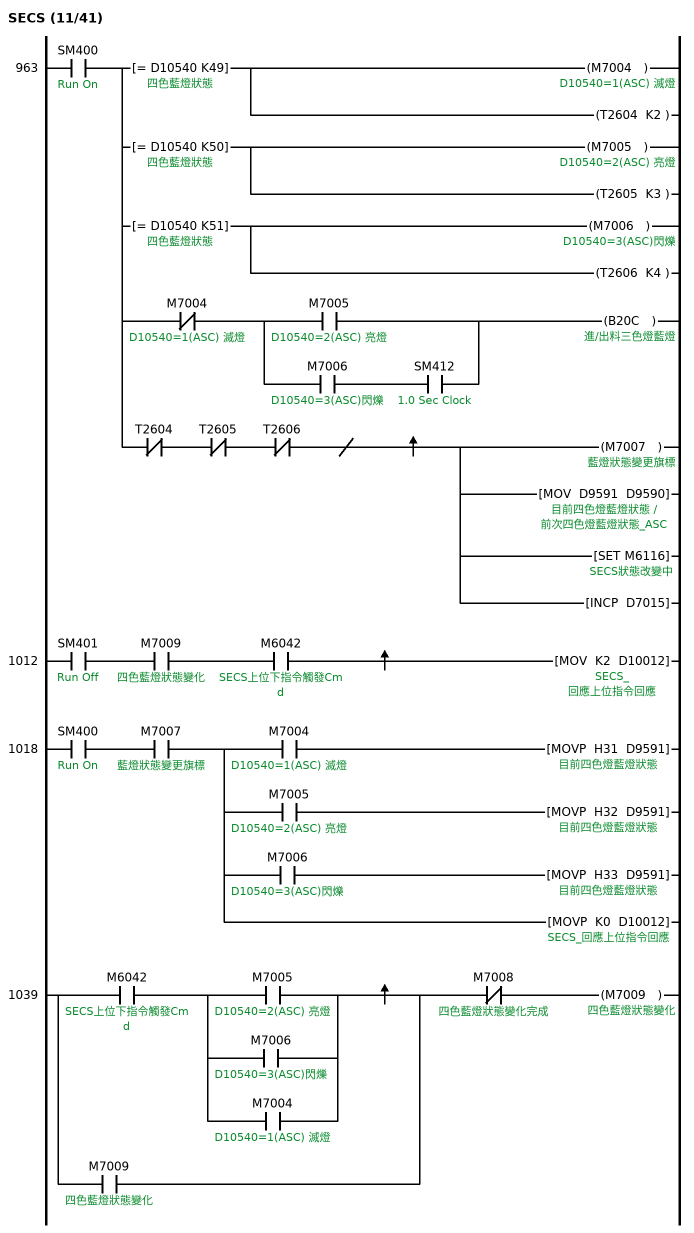
963   LD      SM400  ; Run On
      MPS
      AND=    D10540 K49  ; 四色藍燈狀態
      OUT     M7004  ; D10540=1(ASC) 滅燈
      OUT     T2604 K2
      MRD
      AND=    D10540 K50  ; 四色藍燈狀態
      OUT     M7005  ; D10540=2(ASC) 亮燈
      OUT     T2605 K3
      MRD
      AND=    D10540 K51  ; 四色藍燈狀態
      OUT     M7006  ; D10540=3(ASC)閃爍
      OUT     T2606 K4
      MRD
      ANI     M7004  ; D10540=1(ASC) 滅燈
      LD      M7005  ; D10540=2(ASC) 亮燈
      LD      M7006  ; D10540=3(ASC)閃爍
      AND     SM412  ; 1.0 Sec Clock
      ORB
      ANB
      OUT     B20C  ; 進/出料三色燈藍燈
      MPP
      ANI     T2604
      ANI     T2605
      ANI     T2606
      INV
      MEP
      OUT     M7007  ; 藍燈狀態變更旗標
      MOV     D9591 D9590  ; 目前四色燈藍燈狀態 / 前次四色燈藍燈狀態_ASC
      SET     M6116  ; SECS狀態改變中
      INCP    D7015
1012  LD      SM401  ; Run Off
      AND     M7009  ; 四色藍燈狀態變化
      AND     M6042  ; SECS上位下指令觸發Cmd
      MEP
      MOV     K2 D10012  ; SECS_回應上位指令回應
1018  LD      SM400  ; Run On
      AND     M7007  ; 藍燈狀態變更旗標
      MPS
      AND     M7004  ; D10540=1(ASC) 滅燈
      MOVP    H31 D9591
      MRD
      AND     M7005  ; D10540=2(ASC) 亮燈
      MOVP    H32 D9591
      MRD
      AND     M7006  ; D10540=3(ASC)閃爍
      MOVP    H33 D9591
      MPP
      MOVP    K0 D10012
1039  LD      M6042  ; SECS上位下指令觸發Cmd
      LD      M7005  ; D10540=2(ASC) 亮燈
      OR      M7006  ; D10540=3(ASC)閃爍
      OR      M7004  ; D10540=1(ASC) 滅燈
      ANB
      MEP
      OR      M7009  ; 四色藍燈狀態變化
      ANI     M7008  ; 四色藍燈狀態變化完成
      OUT     M7009  ; 四色藍燈狀態變化
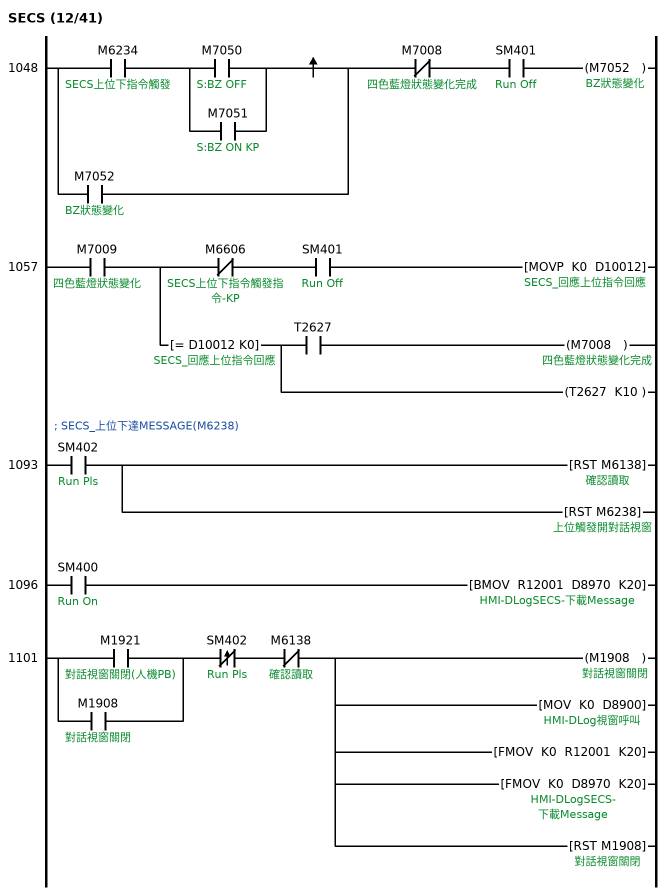
1048  LD      M6234  ; SECS上位下指令觸發
      LD      M7050  ; S:BZ OFF
      OR      M7051  ; S:BZ ON KP
      ANB
      MEP
      OR      M7052  ; BZ狀態變化
      ANI     M7008  ; 四色藍燈狀態變化完成
      AND     SM401  ; Run Off
      OUT     M7052  ; BZ狀態變化
1057  LD      M7009  ; 四色藍燈狀態變化
      MPS
      ANI     M6606  ; SECS上位下指令觸發指令-KP
      AND     SM401  ; Run Off
      MOVP    K0 D10012
      MPP
      AND=    D10012 K0  ; SECS_回應上位指令回應
      MPS
      AND     T2627
      OUT     M7008  ; 四色藍燈狀態變化完成
      MPP
      OUT     T2627 K10
; SECS_上位下達MESSAGE(M6238)
1093  LD      SM402  ; Run Pls
      RST     M6138  ; 確認讀取
      RST     M6238  ; 上位觸發開對話視窗
1096  LD      SM400  ; Run On
      BMOV    R12001 D8970 K20  ; HMI-DLogSECS-下載Message
1101  LD      M1921  ; 對話視窗關閉(人機PB)
      OR      M1908  ; 對話視窗關閉
      ANDPI   SM402  ; Run Pls
      ANI     M6138  ; 確認讀取
      OUT     M1908  ; 對話視窗關閉
      MOV     K0 D8900  ; HMI-DLog視窗呼叫
      FMOV    K0 R12001 K20
      FMOV    K0 D8970 K20
      RST     M1908  ; 對話視窗關閉
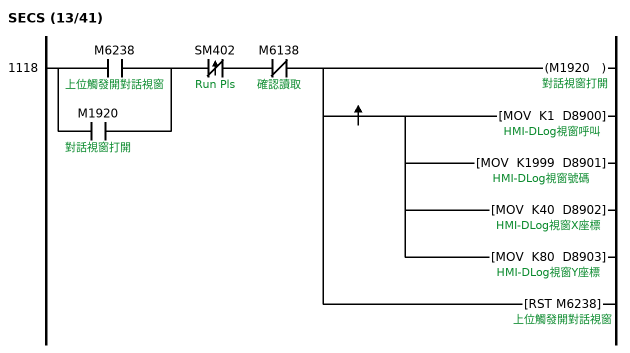
1118  LD      M6238  ; 上位觸發開對話視窗
      OR      M1920  ; 對話視窗打開
      ANDPI   SM402  ; Run Pls
      ANI     M6138  ; 確認讀取
      OUT     M1920  ; 對話視窗打開
      MPS
      MEP
      MOV     K1 D8900
      MOV     K1999 D8901  ; HMI-DLog視窗號碼
      MOV     K40 D8902  ; HMI-DLog視窗X座標
      MOV     K80 D8903  ; HMI-DLog視窗Y座標
      MPP
      RST     M6238  ; 上位觸發開對話視窗
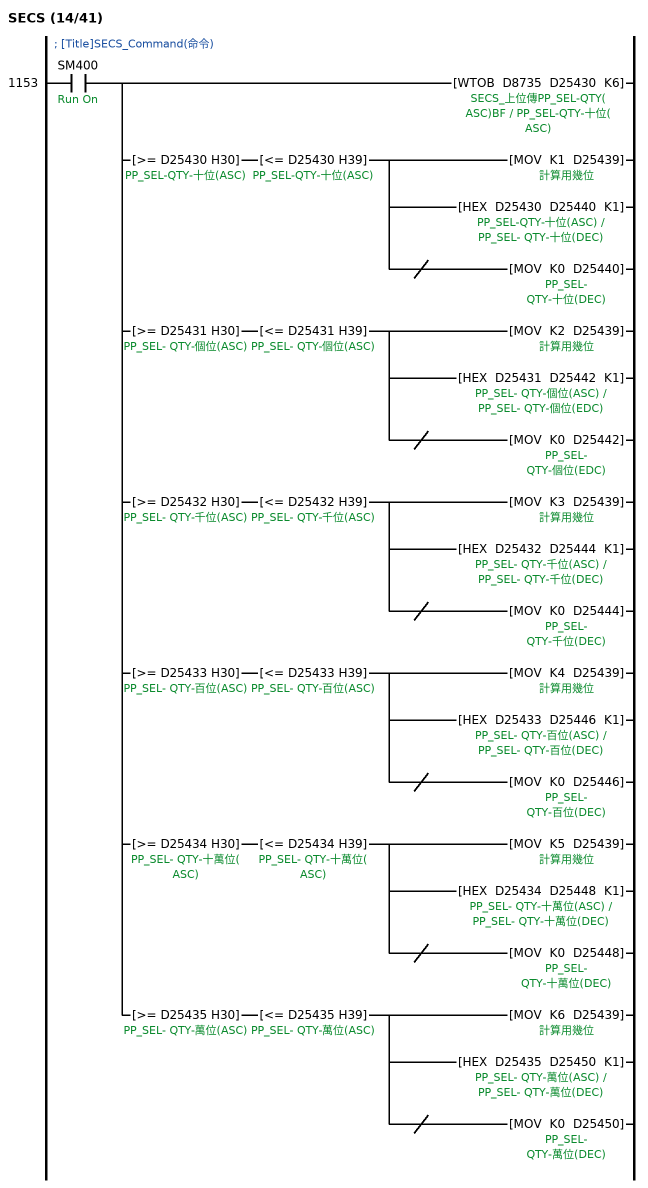
; [Title]SECS_Command(命令)
1153  LD      SM400  ; Run On
      WTOB    D8735 D25430 K6  ; SECS_上位傳PP_SEL-QTY(ASC)BF / PP_SEL-QTY-十位(ASC)
      MPS
      AND>=   D25430 H30  ; PP_SEL-QTY-十位(ASC)
      AND<=   D25430 H39  ; PP_SEL-QTY-十位(ASC)
      MOV     K1 D25439  ; 計算用幾位
      HEX     D25430 D25440 K1  ; PP_SEL- QTY-十位(DEC)
      INV
      MOV     K0 D25440
      MRD
      AND>=   D25431 H30  ; PP_SEL- QTY-個位(ASC)
      AND<=   D25431 H39  ; PP_SEL- QTY-個位(ASC)
      MOV     K2 D25439
      HEX     D25431 D25442 K1  ; PP_SEL- QTY-個位(EDC)
      INV
      MOV     K0 D25442
      MRD
      AND>=   D25432 H30  ; PP_SEL- QTY-千位(ASC)
      AND<=   D25432 H39  ; PP_SEL- QTY-千位(ASC)
      MOV     K3 D25439
      HEX     D25432 D25444 K1  ; PP_SEL- QTY-千位(DEC)
      INV
      MOV     K0 D25444
      MRD
      AND>=   D25433 H30  ; PP_SEL- QTY-百位(ASC)
      AND<=   D25433 H39  ; PP_SEL- QTY-百位(ASC)
      MOV     K4 D25439
      HEX     D25433 D25446 K1  ; PP_SEL- QTY-百位(DEC)
      INV
      MOV     K0 D25446
      MRD
      AND>=   D25434 H30  ; PP_SEL- QTY-十萬位(ASC)
      AND<=   D25434 H39  ; PP_SEL- QTY-十萬位(ASC)
      MOV     K5 D25439
      HEX     D25434 D25448 K1  ; PP_SEL- QTY-十萬位(DEC)
      INV
      MOV     K0 D25448
      MPP
      AND>=   D25435 H30  ; PP_SEL- QTY-萬位(ASC)
      AND<=   D25435 H39  ; PP_SEL- QTY-萬位(ASC)
      MOV     K6 D25439
      HEX     D25435 D25450 K1  ; PP_SEL- QTY-萬位(DEC)
      INV
      MOV     K0 D25450
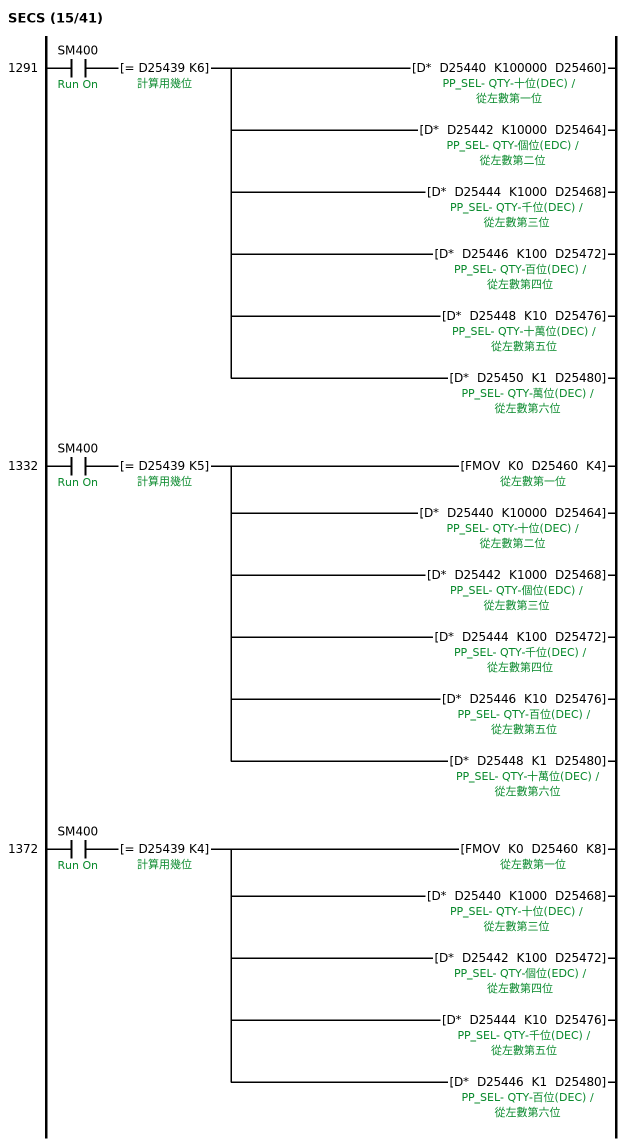
1291  LD      SM400  ; Run On
      AND=    D25439 K6  ; 計算用幾位
      D*      D25440 K100000 D25460  ; 從左數第一位
      D*      D25442 K10000 D25464  ; 從左數第二位
      D*      D25444 K1000 D25468  ; 從左數第三位
      D*      D25446 K100 D25472  ; 從左數第四位
      D*      D25448 K10 D25476  ; 從左數第五位
      D*      D25450 K1 D25480  ; 從左數第六位
1332  LD      SM400  ; Run On
      AND=    D25439 K5  ; 計算用幾位
      FMOV    K0 D25460 K4
      D*      D25440 K10000 D25464
      D*      D25442 K1000 D25468
      D*      D25444 K100 D25472
      D*      D25446 K10 D25476
      D*      D25448 K1 D25480
1372  LD      SM400  ; Run On
      AND=    D25439 K4  ; 計算用幾位
      FMOV    K0 D25460 K8
      D*      D25440 K1000 D25468
      D*      D25442 K100 D25472
      D*      D25444 K10 D25476
      D*      D25446 K1 D25480
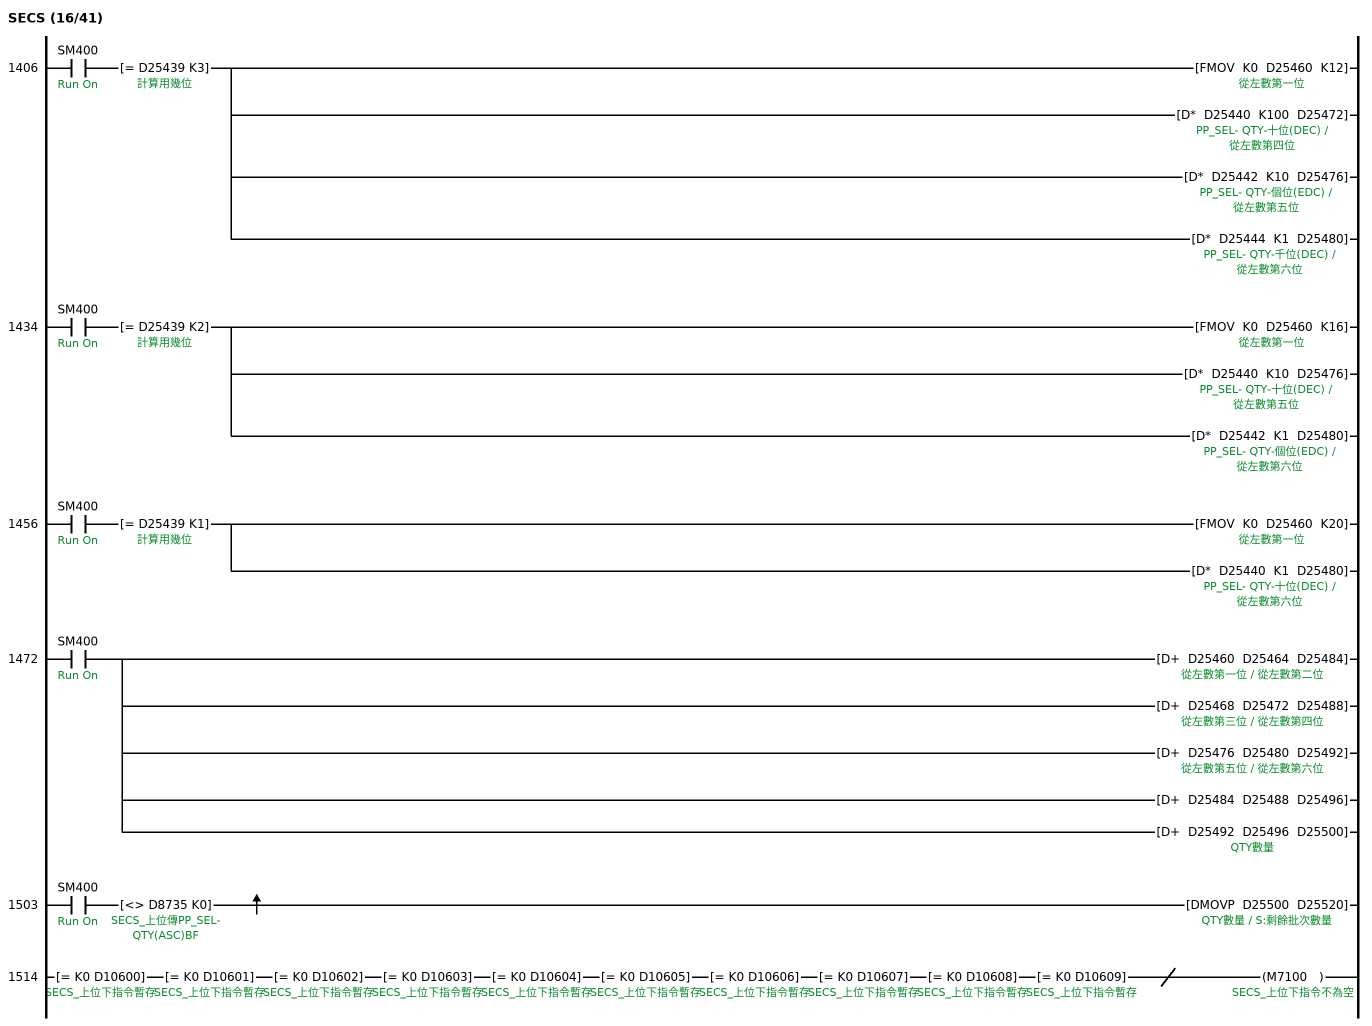
1406  LD      SM400  ; Run On
      AND=    D25439 K3  ; 計算用幾位
      FMOV    K0 D25460 K12
      D*      D25440 K100 D25472
      D*      D25442 K10 D25476
      D*      D25444 K1 D25480
1434  LD      SM400  ; Run On
      AND=    D25439 K2  ; 計算用幾位
      FMOV    K0 D25460 K16
      D*      D25440 K10 D25476
      D*      D25442 K1 D25480
1456  LD      SM400  ; Run On
      AND=    D25439 K1  ; 計算用幾位
      FMOV    K0 D25460 K20
      D*      D25440 K1 D25480
1472  LD      SM400  ; Run On
      D+      D25460 D25464 D25484
      D+      D25468 D25472 D25488
      D+      D25476 D25480 D25492
      D+      D25484 D25488 D25496
      D+      D25492 D25496 D25500  ; QTY數量
1503  LD      SM400  ; Run On
      AND<>   D8735 K0  ; SECS_上位傳PP_SEL-QTY(ASC)BF
      MEP
      DMOVP   D25500 D25520  ; S:剩餘批次數量
1514  LD=     K0 D10600  ; SECS_上位下指令暫存
      AND=    K0 D10601  ; SECS_上位下指令暫存
      AND=    K0 D10602  ; SECS_上位下指令暫存
      AND=    K0 D10603  ; SECS_上位下指令暫存
      AND=    K0 D10604  ; SECS_上位下指令暫存
      AND=    K0 D10605  ; SECS_上位下指令暫存
      AND=    K0 D10606  ; SECS_上位下指令暫存
      AND=    K0 D10607  ; SECS_上位下指令暫存
      AND=    K0 D10608  ; SECS_上位下指令暫存
      AND=    K0 D10609  ; SECS_上位下指令暫存
      INV
      OUT     M7100  ; SECS_上位下指令不為空
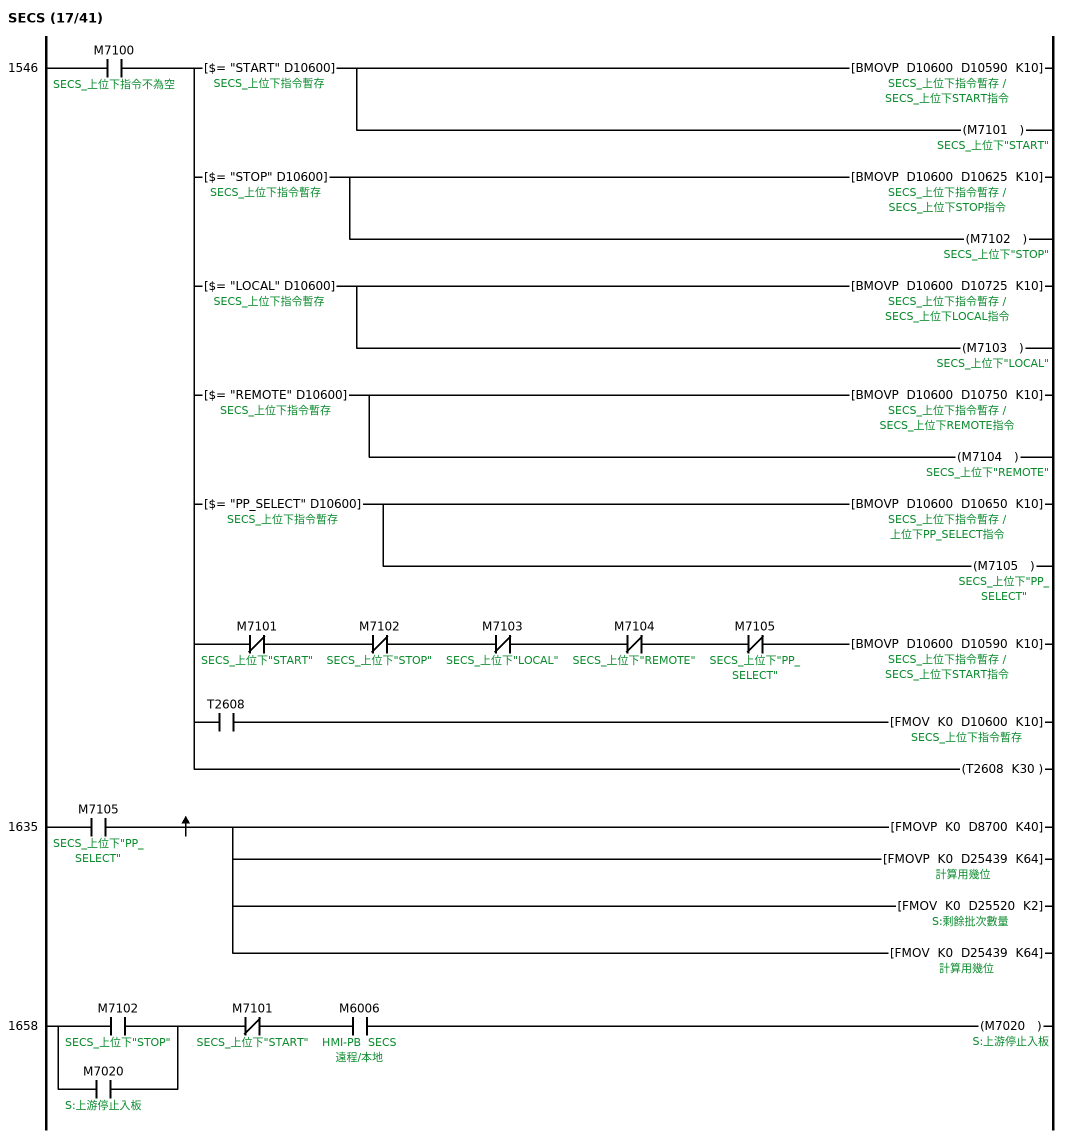
1546  LD      M7100  ; SECS_上位下指令不為空
      MPS
      AND$=   "START" D10600  ; SECS_上位下指令暫存
      BMOVP   D10600 D10590 K10  ; SECS_上位下START指令
      OUT     M7101  ; SECS_上位下"START"
      MRD
      AND$=   "STOP" D10600  ; SECS_上位下指令暫存
      BMOVP   D10600 D10625 K10  ; SECS_上位下STOP指令
      OUT     M7102  ; SECS_上位下"STOP"
      MRD
      AND$=   "LOCAL" D10600  ; SECS_上位下指令暫存
      BMOVP   D10600 D10725 K10  ; SECS_上位下LOCAL指令
      OUT     M7103  ; SECS_上位下"LOCAL"
      MRD
      AND$=   "REMOTE" D10600  ; SECS_上位下指令暫存
      BMOVP   D10600 D10750 K10  ; SECS_上位下REMOTE指令
      OUT     M7104  ; SECS_上位下"REMOTE"
      MRD
      AND$=   "PP_SELECT" D10600  ; SECS_上位下指令暫存
      BMOVP   D10600 D10650 K10  ; 上位下PP_SELECT指令
      OUT     M7105  ; SECS_上位下"PP_SELECT"
      MRD
      ANI     M7101  ; SECS_上位下"START"
      ANI     M7102  ; SECS_上位下"STOP"
      ANI     M7103  ; SECS_上位下"LOCAL"
      ANI     M7104  ; SECS_上位下"REMOTE"
      ANI     M7105  ; SECS_上位下"PP_SELECT"
      BMOVP   D10600 D10590 K10
      MRD
      AND     T2608
      FMOV    K0 D10600 K10
      MPP
      OUT     T2608 K30
1635  LD      M7105  ; SECS_上位下"PP_SELECT"
      MEP
      FMOVP   K0 D8700 K40
      FMOVP   K0 D25439 K64
      FMOV    K0 D25520 K2
      FMOV    K0 D25439 K64
1658  LD      M7102  ; SECS_上位下"STOP"
      OR      M7020  ; S:上游停止入板
      ANI     M7101  ; SECS_上位下"START"
      AND     M6006  ; HMI-PB  SECS  遠程/本地
      OUT     M7020  ; S:上游停止入板
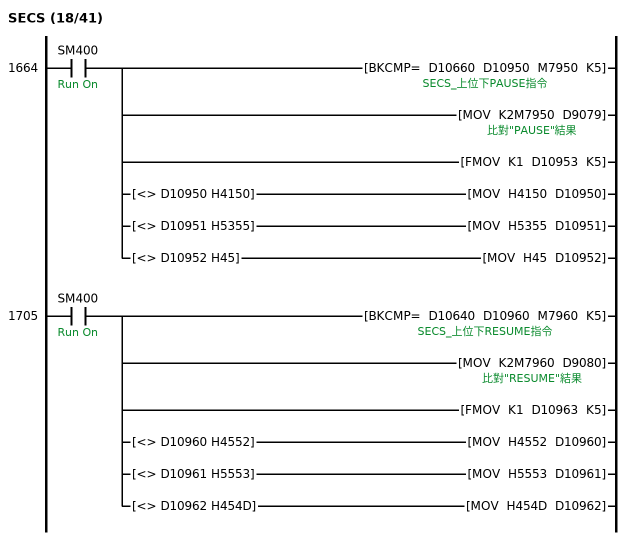
1664  LD      SM400  ; Run On
      BKCMP=  D10660 D10950 M7950 K5  ; SECS_上位下PAUSE指令
        [note] 上位下PAUSE指令
      MOV     K2M7950 D9079  ; 比對"PAUSE"結果
      FMOV    K1 D10953 K5
      MPS
      AND<>   D10950 H4150
      MOV     H4150 D10950
      MRD
      AND<>   D10951 H5355
      MOV     H5355 D10951
      MPP
      AND<>   D10952 H45
      MOV     H45 D10952
1705  LD      SM400  ; Run On
      BKCMP=  D10640 D10960 M7960 K5  ; SECS_上位下RESUME指令
        [note] 上位下RESUME指令
      MOV     K2M7960 D9080  ; 比對"RESUME"結果
      FMOV    K1 D10963 K5
      MPS
      AND<>   D10960 H4552
      MOV     H4552 D10960
      MRD
      AND<>   D10961 H5553
      MOV     H5553 D10961
      MPP
      AND<>   D10962 H454D
      MOV     H454D D10962
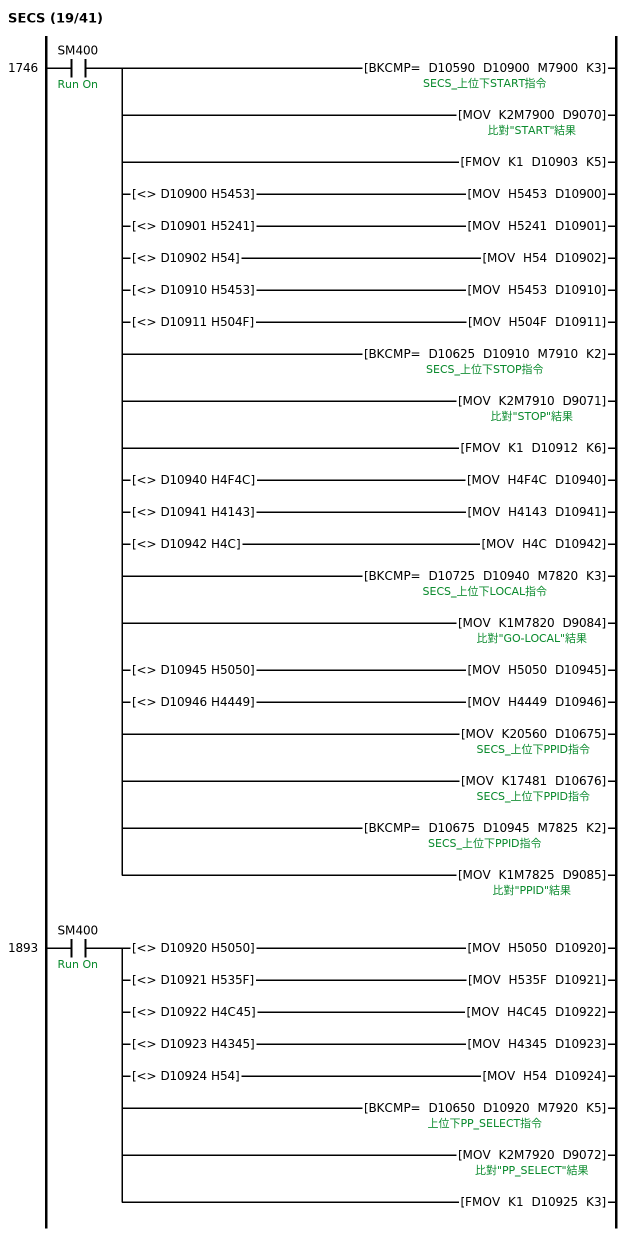
1746  LD      SM400  ; Run On
      BKCMP=  D10590 D10900 M7900 K3
        [note] 上位下START指令
      MOV     K2M7900 D9070  ; 比對"START"結果
      FMOV    K1 D10903 K5
      MPS
      AND<>   D10900 H5453
      MOV     H5453 D10900
      MRD
      AND<>   D10901 H5241
      MOV     H5241 D10901
      MRD
      AND<>   D10902 H54
      MOV     H54 D10902
      MRD
      AND<>   D10910 H5453
      MOV     H5453 D10910
      MRD
      AND<>   D10911 H504F
      MOV     H504F D10911
      MPP
      BKCMP=  D10625 D10910 M7910 K2
        [note] 上位下STOP指令
      MOV     K2M7910 D9071  ; 比對"STOP"結果
      FMOV    K1 D10912 K6
      MPS
      AND<>   D10940 H4F4C
      MOV     H4F4C D10940
      MRD
      AND<>   D10941 H4143
      MOV     H4143 D10941
      MRD
      AND<>   D10942 H4C
      MOV     H4C D10942
      MPP
      BKCMP=  D10725 D10940 M7820 K3
        [note] 上位下GO-LOCAL指令
      MOV     K1M7820 D9084  ; 比對"GO-LOCAL"結果
      MPS
      AND<>   D10945 H5050
      MOV     H5050 D10945
      MRD
      AND<>   D10946 H4449
      MOV     H4449 D10946
      MPP
      MOV     K20560 D10675  ; SECS_上位下PPID指令
      MOV     K17481 D10676  ; SECS_上位下PPID指令
      BKCMP=  D10675 D10945 M7825 K2
        [note] 上位下PPID指令
      MOV     K1M7825 D9085  ; 比對"PPID"結果
1893  LD      SM400  ; Run On
      MPS
      AND<>   D10920 H5050
      MOV     H5050 D10920
      MRD
      AND<>   D10921 H535F
      MOV     H535F D10921
      MRD
      AND<>   D10922 H4C45
      MOV     H4C45 D10922
      MRD
      AND<>   D10923 H4345
      MOV     H4345 D10923
      MRD
      AND<>   D10924 H54
      MOV     H54 D10924
      MPP
      BKCMP=  D10650 D10920 M7920 K5
        [note] 上位下PP_SELECT指令
      MOV     K2M7920 D9072  ; 比對"PP_SELECT"結果
      FMOV    K1 D10925 K3
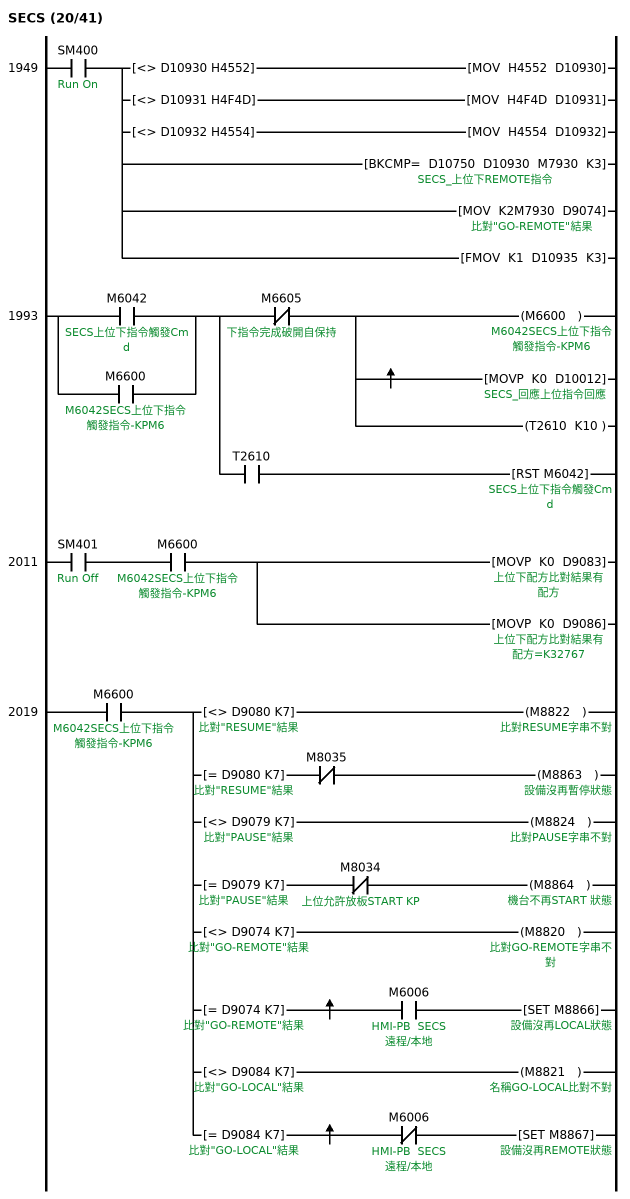
1949  LD      SM400  ; Run On
      MPS
      AND<>   D10930 H4552
      MOV     H4552 D10930
      MRD
      AND<>   D10931 H4F4D
      MOV     H4F4D D10931
      MRD
      AND<>   D10932 H4554
      MOV     H4554 D10932
      MPP
      BKCMP=  D10750 D10930 M7930 K3
        [note] 上位下GO-REMOTE指令
      MOV     K2M7930 D9074  ; 比對"GO-REMOTE"結果
      FMOV    K1 D10935 K3
1993  LD      M6042  ; SECS上位下指令觸發Cmd
      OR      M6600  ; M6042SECS上位下指令觸發指令-KPM6
      MPS
      ANI     M6605  ; 下指令完成破開自保持
      OUT     M6600  ; M6042SECS上位下指令觸發指令-KPM6
      MPS
      MEP
      MOVP    K0 D10012
      MPP
      OUT     T2610 K10
      MPP
      AND     T2610
      RST     M6042  ; SECS上位下指令觸發Cmd
2011  LD      SM401  ; Run Off
      AND     M6600  ; M6042SECS上位下指令觸發指令-KPM6
      MOVP    K0 D9083  ; 上位下配方比對結果有配方
      MOVP    K0 D9086  ; 上位下配方比對結果有配方=K32767
2019  LD      M6600  ; M6042SECS上位下指令觸發指令-KPM6
      MPS
      AND<>   D9080 K7  ; 比對"RESUME"結果
      OUT     M8822  ; 比對RESUME字串不對
      MRD
      AND=    D9080 K7  ; 比對"RESUME"結果
      ANI     M8035
      OUT     M8863  ; 設備沒再暫停狀態
      MRD
      AND<>   D9079 K7  ; 比對"PAUSE"結果
      OUT     M8824  ; 比對PAUSE字串不對
      MRD
      AND=    D9079 K7  ; 比對"PAUSE"結果
      ANI     M8034  ; 上位允許放板START KP
      OUT     M8864  ; 機台不再START 狀態
      MRD
      AND<>   D9074 K7  ; 比對"GO-REMOTE"結果
      OUT     M8820  ; 比對GO-REMOTE字串不對
      MRD
      AND=    D9074 K7  ; 比對"GO-REMOTE"結果
      MEP
      AND     M6006  ; HMI-PB  SECS  遠程/本地
      SET     M8866  ; 設備沒再LOCAL狀態
      MRD
      AND<>   D9084 K7  ; 比對"GO-LOCAL"結果
      OUT     M8821  ; 名稱GO-LOCAL比對不對
      MPP
      AND=    D9084 K7  ; 比對"GO-LOCAL"結果
      MEP
      ANI     M6006  ; HMI-PB  SECS  遠程/本地
      SET     M8867  ; 設備沒再REMOTE狀態
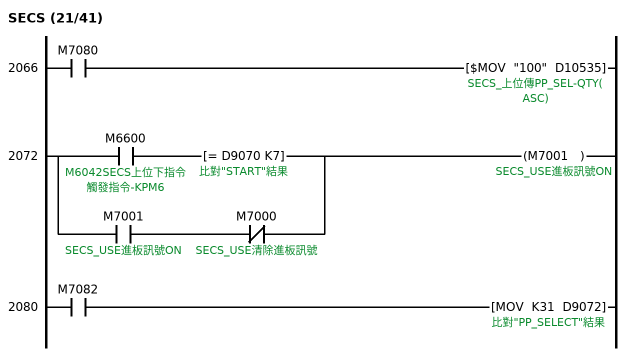
2066  LD      M7080
      $MOV    "100" D10535  ; SECS_上位傳PP_SEL-QTY(ASC)
2072  LD      M6600  ; M6042SECS上位下指令觸發指令-KPM6
      AND=    D9070 K7  ; 比對"START"結果
      LD      M7001  ; SECS_USE進板訊號ON
      ANI     M7000  ; SECS_USE清除進板訊號
      ORB
      OUT     M7001  ; SECS_USE進板訊號ON
2080  LD      M7082
      MOV     K31 D9072
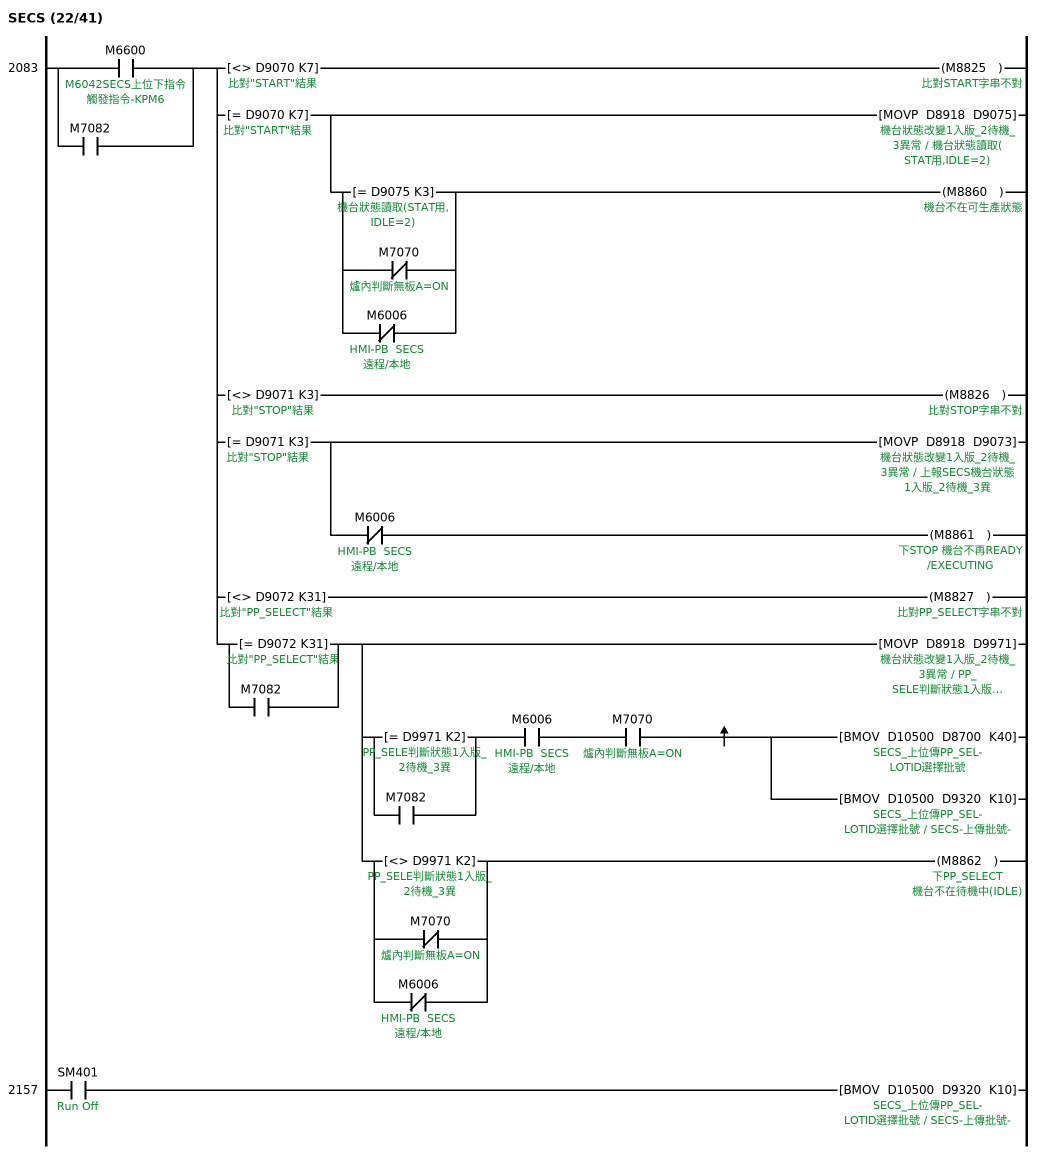
2083  LD      M6600  ; M6042SECS上位下指令觸發指令-KPM6
      OR      M7082
      MPS
      AND<>   D9070 K7  ; 比對"START"結果
      OUT     M8825  ; 比對START字串不對
      MRD
      AND=    D9070 K7  ; 比對"START"結果
      MOVP    D8918 D9075  ; 機台狀態讀取(STAT用,IDLE=2)
      LD=     D9075 K3  ; 機台狀態讀取(STAT用,IDLE=2)
      ORI     M7070  ; 爐內判斷無板A=ON
      ORI     M6006  ; HMI-PB  SECS  遠程/本地
      ANB
      OUT     M8860  ; 機台不在可生產狀態
      MRD
      AND<>   D9071 K3  ; 比對"STOP"結果
      OUT     M8826  ; 比對STOP字串不對
      MRD
      AND=    D9071 K3  ; 比對"STOP"結果
      MOVP    D8918 D9073  ; 上報SECS機台狀態1入版_2待機_3異
      ANI     M6006  ; HMI-PB  SECS  遠程/本地
      OUT     M8861  ; 下STOP 機台不再READY/EXECUTING
      MRD
      AND<>   D9072 K31  ; 比對"PP_SELECT"結果
      OUT     M8827  ; 比對PP_SELECT字串不對
      MPP
      LD=     D9072 K31  ; 比對"PP_SELECT"結果
      OR      M7082
      ANB
      MOVP    D8918 D9971  ; PP_SELE判斷狀態1入版_2待機_3異
      MPS
      LD=     D9971 K2  ; PP_SELE判斷狀態1入版_2待機_3異
      OR      M7082
      ANB
      AND     M6006  ; HMI-PB  SECS  遠程/本地
      AND     M7070  ; 爐內判斷無板A=ON
      MEP
      BMOV    D10500 D8700 K40  ; SECS_上位傳PP_SEL-LOTID選擇批號
      BMOV    D10500 D9320 K10  ; SECS-上傳批號-
      MPP
      LD<>    D9971 K2  ; PP_SELE判斷狀態1入版_2待機_3異
      ORI     M7070  ; 爐內判斷無板A=ON
      ORI     M6006  ; HMI-PB  SECS  遠程/本地
      ANB
      OUT     M8862  ; 下PP_SELECT 機台不在待機中(IDLE)
2157  LD      SM401  ; Run Off
      BMOV    D10500 D9320 K10
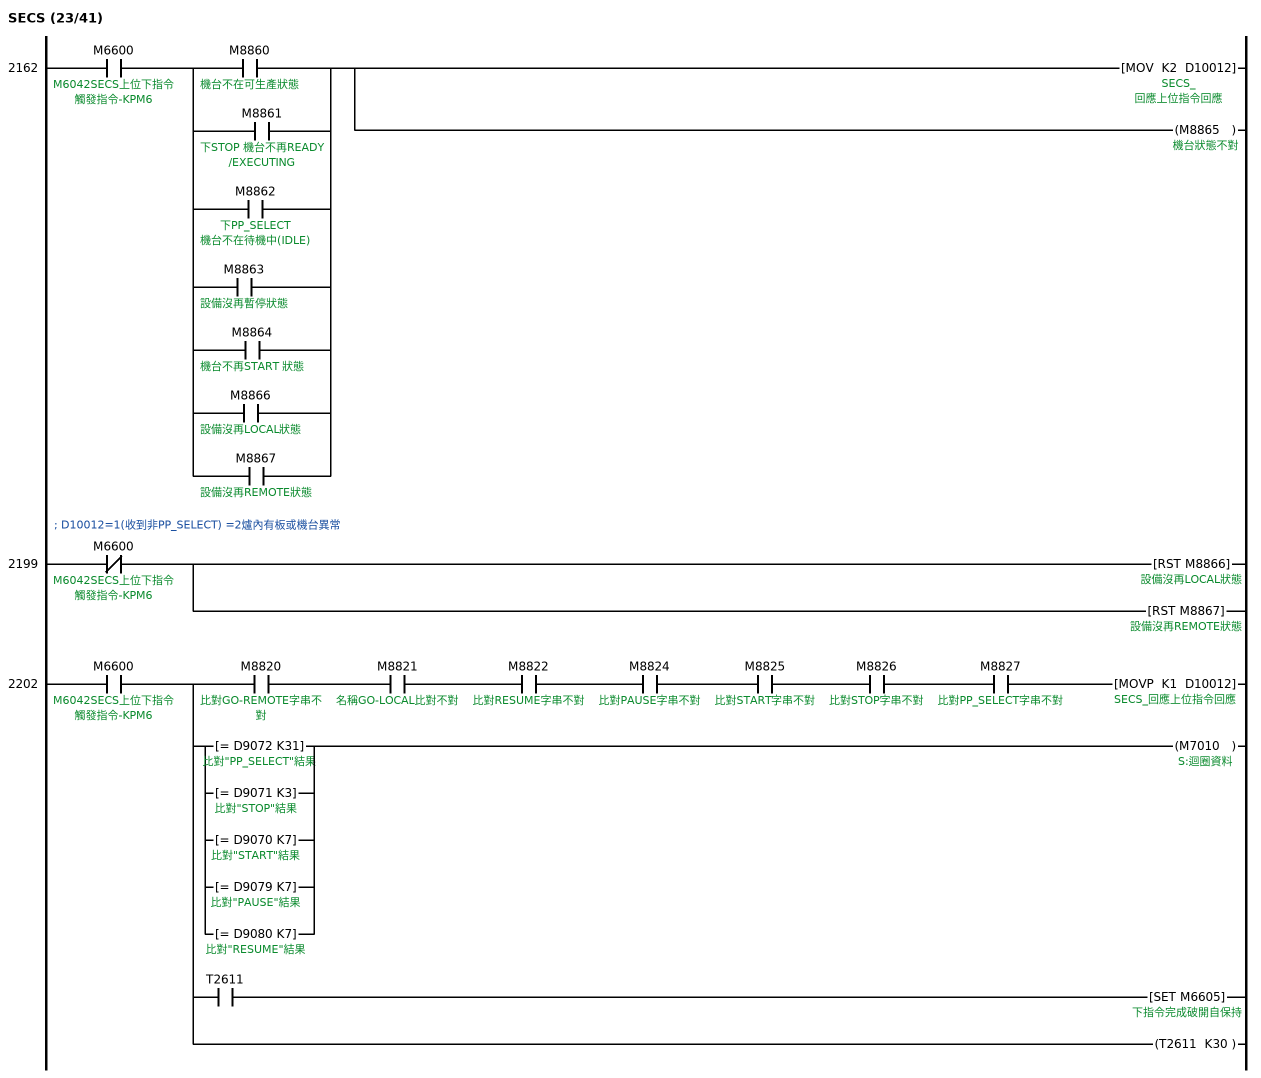
2162  LD      M6600  ; M6042SECS上位下指令觸發指令-KPM6
      LD      M8860  ; 機台不在可生產狀態
      OR      M8861  ; 下STOP 機台不再READY/EXECUTING
      OR      M8862  ; 下PP_SELECT 機台不在待機中(IDLE)
      OR      M8863  ; 設備沒再暫停狀態
      OR      M8864  ; 機台不再START 狀態
      OR      M8866  ; 設備沒再LOCAL狀態
      OR      M8867  ; 設備沒再REMOTE狀態
      ANB
      MOV     K2 D10012
      OUT     M8865  ; 機台狀態不對
; D10012=1(收到非PP_SELECT) =2爐內有板或機台異常
2199  LDI     M6600  ; M6042SECS上位下指令觸發指令-KPM6
      RST     M8866  ; 設備沒再LOCAL狀態
      RST     M8867  ; 設備沒再REMOTE狀態
2202  LD      M6600  ; M6042SECS上位下指令觸發指令-KPM6
      MPS
      AND     M8820  ; 比對GO-REMOTE字串不對
      AND     M8821  ; 名稱GO-LOCAL比對不對
      AND     M8822  ; 比對RESUME字串不對
      AND     M8824  ; 比對PAUSE字串不對
      AND     M8825  ; 比對START字串不對
      AND     M8826  ; 比對STOP字串不對
      AND     M8827  ; 比對PP_SELECT字串不對
      MOVP    K1 D10012
      MRD
      LD=     D9072 K31  ; 比對"PP_SELECT"結果
      OR=     D9071 K3  ; 比對"STOP"結果
      OR=     D9070 K7  ; 比對"START"結果
      OR=     D9079 K7  ; 比對"PAUSE"結果
      OR=     D9080 K7  ; 比對"RESUME"結果
      ANB
      OUT     M7010  ; S:迴圈資料
      MRD
      AND     T2611
      SET     M6605  ; 下指令完成破開自保持
      MPP
      OUT     T2611 K30
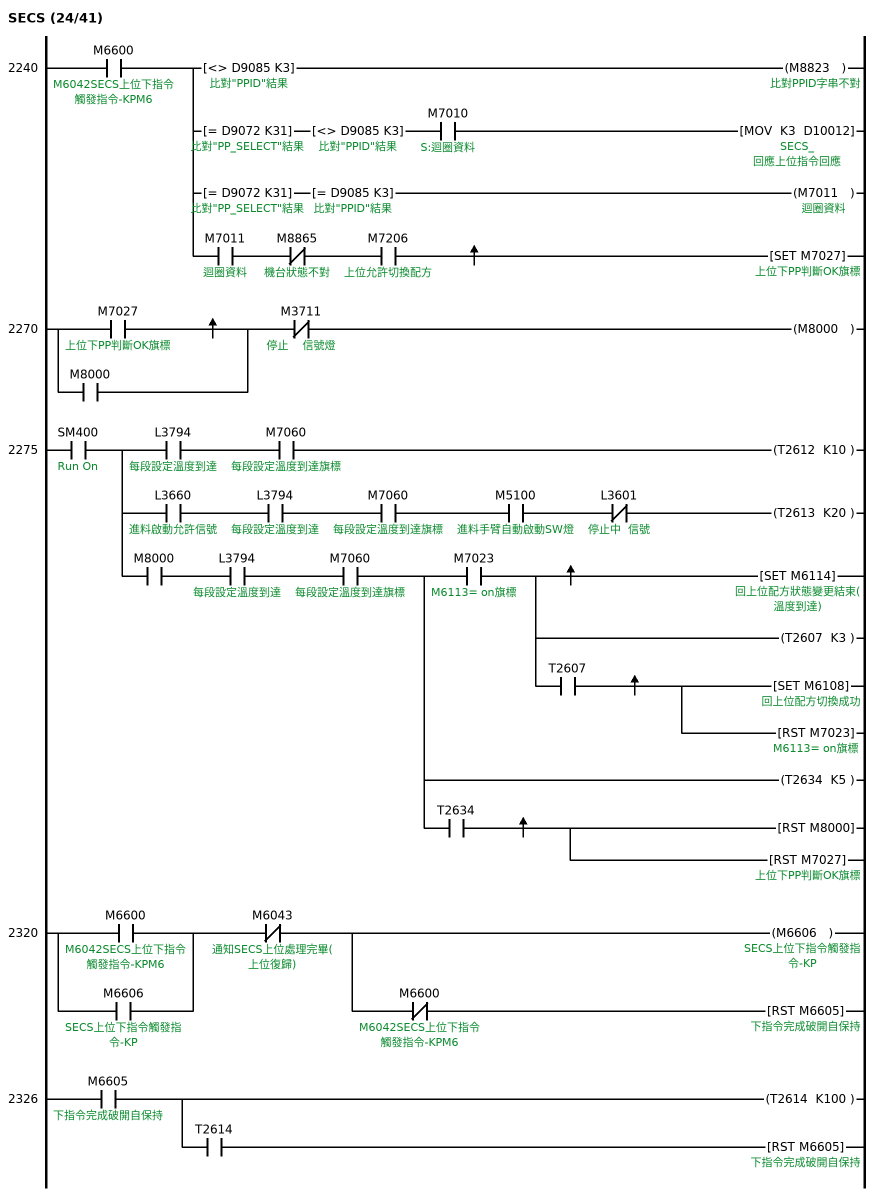
2240  LD      M6600  ; M6042SECS上位下指令觸發指令-KPM6
      MPS
      AND<>   D9085 K3  ; 比對"PPID"結果
      OUT     M8823  ; 比對PPID字串不對
      MRD
      AND=    D9072 K31  ; 比對"PP_SELECT"結果
      AND<>   D9085 K3  ; 比對"PPID"結果
      AND     M7010  ; S:迴圈資料
      MOV     K3 D10012
      MRD
      AND=    D9072 K31  ; 比對"PP_SELECT"結果
      AND=    D9085 K3  ; 比對"PPID"結果
      OUT     M7011  ; 迴圈資料
      MPP
      AND     M7011  ; 迴圈資料
      ANI     M8865  ; 機台狀態不對
      AND     M7206  ; 上位允許切換配方
      MEP
      SET     M7027  ; 上位下PP判斷OK旗標
2270  LD      M7027  ; 上位下PP判斷OK旗標
      MEP
      OR      M8000
      ANI     M3711  ; 停止    信號燈
      OUT     M8000
2275  LD      SM400  ; Run On
      MPS
      AND     L3794  ; 每段設定溫度到達
      AND     M7060  ; 每段設定溫度到達旗標
      OUT     T2612 K10
      MRD
      AND     L3660  ; 進料啟動允許信號
      AND     L3794  ; 每段設定溫度到達
      AND     M7060  ; 每段設定溫度到達旗標
      AND     M5100  ; 進料手臂自動啟動SW燈
      ANI     L3601  ; 停止中  信號
      OUT     T2613 K20
      MPP
      AND     M8000
      AND     L3794  ; 每段設定溫度到達
      AND     M7060  ; 每段設定溫度到達旗標
      MPS
      AND     M7023  ; M6113= on旗標
      MPS
      MEP
      SET     M6114  ; 回上位配方狀態變更結束(溫度到達)
      MPP
      OUT     T2607 K3
      AND     T2607
      MEP
      SET     M6108  ; 回上位配方切換成功
      RST     M7023  ; M6113= on旗標
      MPP
      OUT     T2634 K5
      AND     T2634
      MEP
      RST     M8000
      RST     M7027  ; 上位下PP判斷OK旗標
2320  LD      M6600  ; M6042SECS上位下指令觸發指令-KPM6
      OR      M6606  ; SECS上位下指令觸發指令-KP
      ANI     M6043  ; 通知SECS上位處理完畢(上位復歸)
      OUT     M6606  ; SECS上位下指令觸發指令-KP
      ANI     M6600  ; M6042SECS上位下指令觸發指令-KPM6
      RST     M6605  ; 下指令完成破開自保持
2326  LD      M6605  ; 下指令完成破開自保持
      OUT     T2614 K100
      AND     T2614
      RST     M6605  ; 下指令完成破開自保持
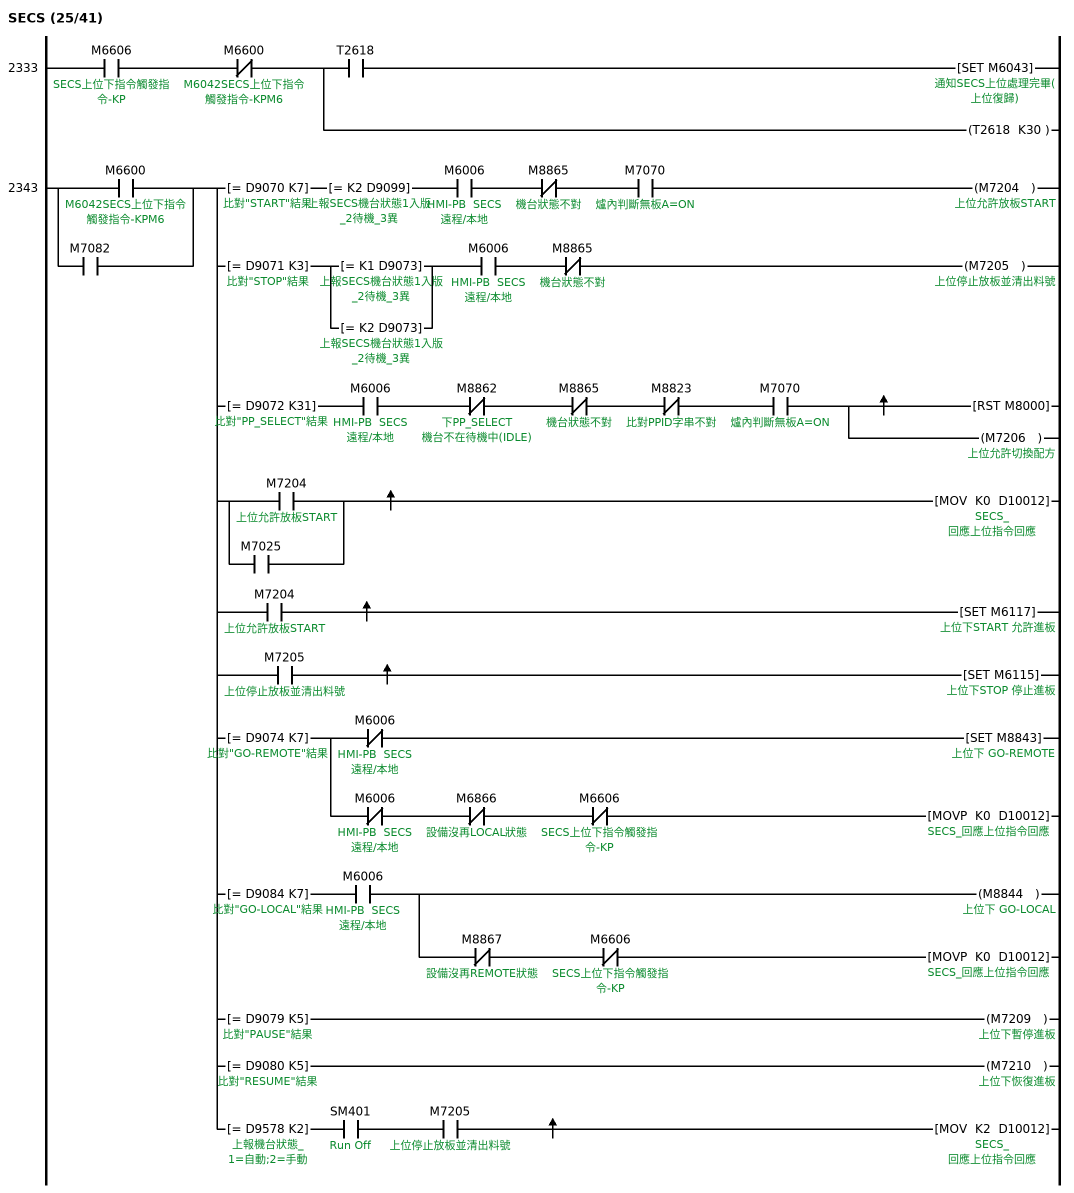
2333  LD      M6606  ; SECS上位下指令觸發指令-KP
      ANI     M6600  ; M6042SECS上位下指令觸發指令-KPM6
      MPS
      AND     T2618
      SET     M6043  ; 通知SECS上位處理完畢(上位復歸)
      MPP
      OUT     T2618 K30
2343  LD      M6600  ; M6042SECS上位下指令觸發指令-KPM6
      OR      M7082
      MPS
      AND=    D9070 K7  ; 比對"START"結果
      AND=    K2 D9099  ; 上報SECS機台狀態1入版_2待機_3異
      AND     M6006  ; HMI-PB  SECS  遠程/本地
      ANI     M8865  ; 機台狀態不對
      AND     M7070  ; 爐內判斷無板A=ON
      OUT     M7204  ; 上位允許放板START
      MRD
      AND=    D9071 K3  ; 比對"STOP"結果
      LD=     K1 D9073  ; 上報SECS機台狀態1入版_2待機_3異
      OR=     K2 D9073  ; 上報SECS機台狀態1入版_2待機_3異
      ANB
      AND     M6006  ; HMI-PB  SECS  遠程/本地
      ANI     M8865  ; 機台狀態不對
      OUT     M7205  ; 上位停止放板並清出料號
      MRD
      AND=    D9072 K31  ; 比對"PP_SELECT"結果
      AND     M6006  ; HMI-PB  SECS  遠程/本地
      ANI     M8862  ; 下PP_SELECT 機台不在待機中(IDLE)
      ANI     M8865  ; 機台狀態不對
      ANI     M8823  ; 比對PPID字串不對
      AND     M7070  ; 爐內判斷無板A=ON
      MPS
      MEP
      RST     M8000
      MPP
      OUT     M7206  ; 上位允許切換配方
      MRD
      LD      M7204  ; 上位允許放板START
      OR      M7025
      ANB
      MEP
      MOV     K0 D10012
      MRD
      AND     M7204  ; 上位允許放板START
      MEP
      SET     M6117  ; 上位下START 允許進板
      MRD
      AND     M7205  ; 上位停止放板並清出料號
      MEP
      SET     M6115  ; 上位下STOP 停止進板
      MRD
      AND=    D9074 K7  ; 比對"GO-REMOTE"結果
      MPS
      ANI     M6006  ; HMI-PB  SECS  遠程/本地
      SET     M8843  ; 上位下 GO-REMOTE
      MPP
      ANI     M6006  ; HMI-PB  SECS  遠程/本地
      ANI     M6866  ; 設備沒再LOCAL狀態
      ANI     M6606  ; SECS上位下指令觸發指令-KP
      MOVP    K0 D10012
      MRD
      AND=    D9084 K7  ; 比對"GO-LOCAL"結果
      AND     M6006  ; HMI-PB  SECS  遠程/本地
      OUT     M8844  ; 上位下 GO-LOCAL
      ANI     M8867  ; 設備沒再REMOTE狀態
      ANI     M6606  ; SECS上位下指令觸發指令-KP
      MOVP    K0 D10012
      MRD
      AND=    D9079 K5  ; 比對"PAUSE"結果
      OUT     M7209  ; 上位下暫停進板
      MRD
      AND=    D9080 K5  ; 比對"RESUME"結果
      OUT     M7210  ; 上位下恢復進板
      MPP
      AND=    D9578 K2  ; 上報機台狀態_1=自動;2=手動
      AND     SM401  ; Run Off
      AND     M7205  ; 上位停止放板並清出料號
      MEP
      MOV     K2 D10012
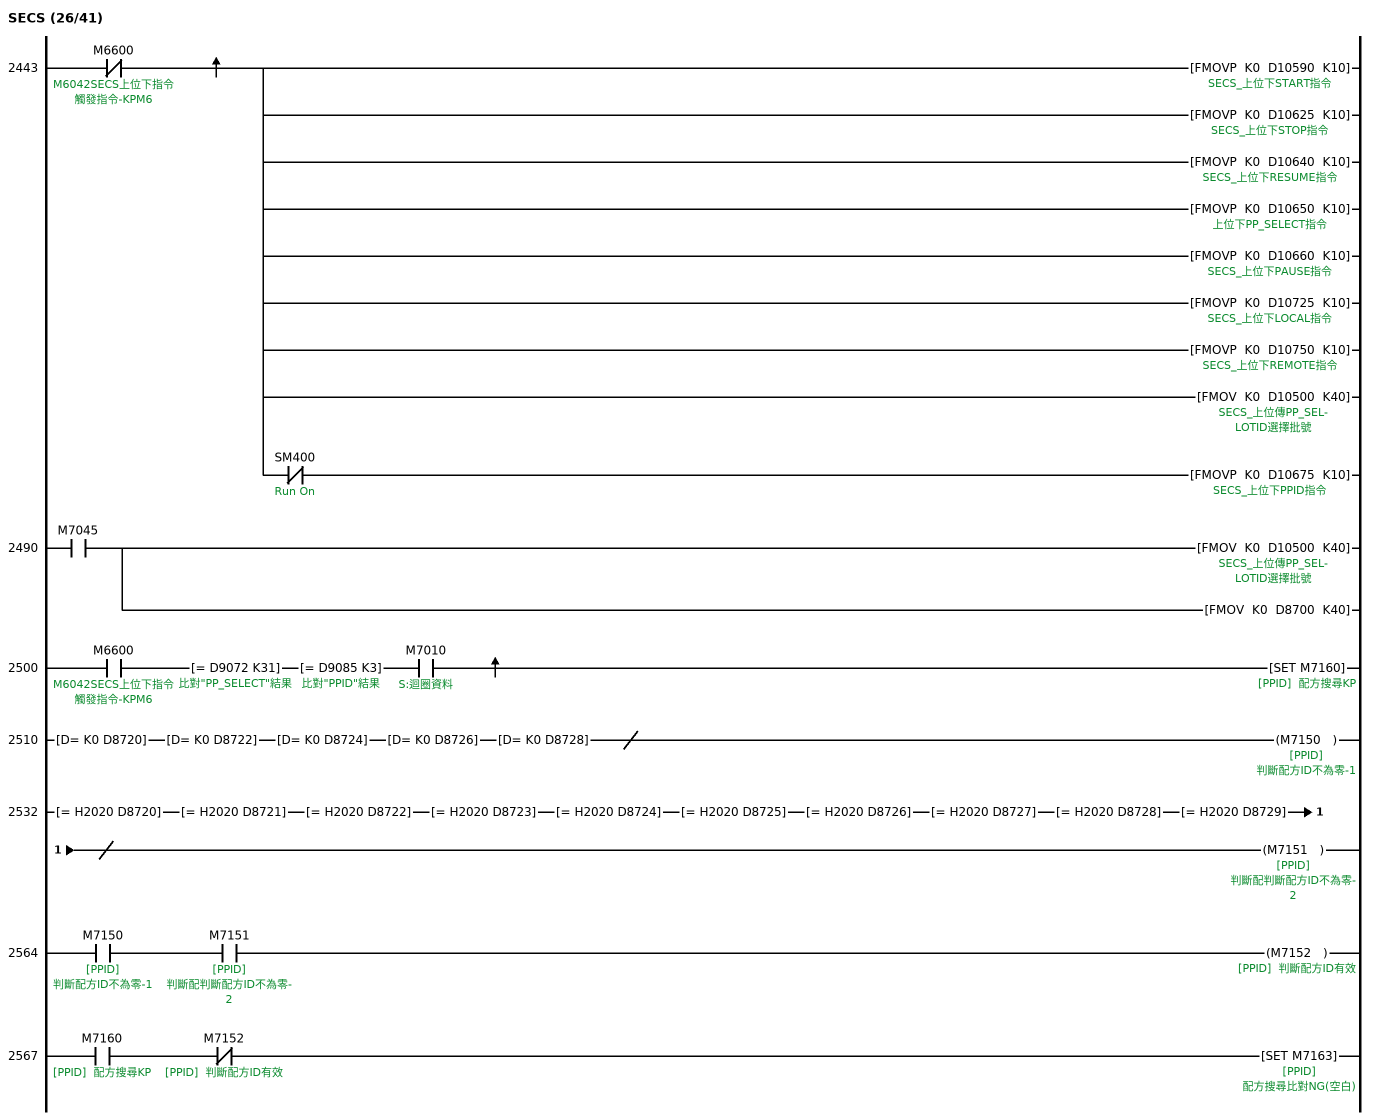
2443  LDI     M6600  ; M6042SECS上位下指令觸發指令-KPM6
      MEP
      FMOVP   K0 D10590 K10
      FMOVP   K0 D10625 K10
      FMOVP   K0 D10640 K10
      FMOVP   K0 D10650 K10
      FMOVP   K0 D10660 K10
      FMOVP   K0 D10725 K10
      FMOVP   K0 D10750 K10
      FMOV    K0 D10500 K40
      ANI     SM400  ; Run On
      FMOVP   K0 D10675 K10
2490  LD      M7045
      FMOV    K0 D10500 K40
      FMOV    K0 D8700 K40
2500  LD      M6600  ; M6042SECS上位下指令觸發指令-KPM6
      AND=    D9072 K31  ; 比對"PP_SELECT"結果
      AND=    D9085 K3  ; 比對"PPID"結果
      AND     M7010  ; S:迴圈資料
      MEP
      SET     M7160  ; [PPID]  配方搜尋KP
2510  LDD=    K0 D8720
      ANDD=   K0 D8722
      ANDD=   K0 D8724
      ANDD=   K0 D8726
      ANDD=   K0 D8728
      INV
      OUT     M7150  ; [PPID]  判斷配方ID不為零-1
2532  LD=     H2020 D8720
      AND=    H2020 D8721
      AND=    H2020 D8722
      AND=    H2020 D8723
      AND=    H2020 D8724
      AND=    H2020 D8725
      AND=    H2020 D8726
      AND=    H2020 D8727
      AND=    H2020 D8728
      AND=    H2020 D8729
      INV
      OUT     M7151  ; [PPID]  判斷配判斷配方ID不為零-2
2564  LD      M7150  ; [PPID]  判斷配方ID不為零-1
      AND     M7151  ; [PPID]  判斷配判斷配方ID不為零-2
      OUT     M7152  ; [PPID]  判斷配方ID有效
2567  LD      M7160  ; [PPID]  配方搜尋KP
      ANI     M7152  ; [PPID]  判斷配方ID有效
      SET     M7163  ; [PPID]  配方搜尋比對NG(空白)
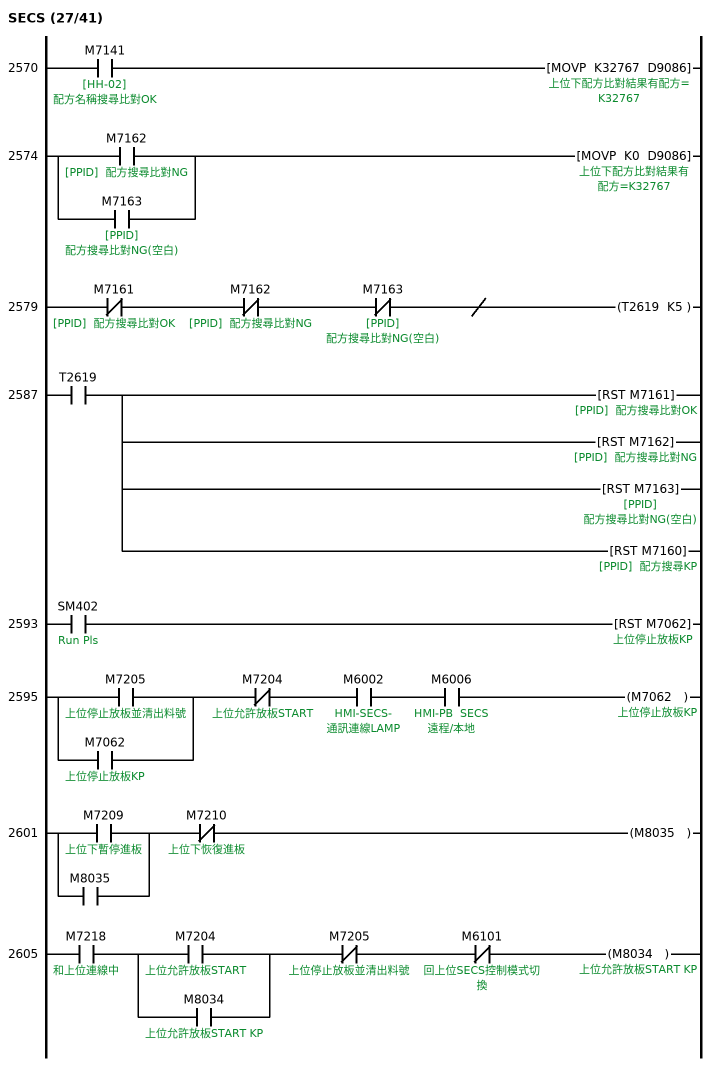
2570  LD      M7141  ; [HH-02] 配方名稱搜尋比對OK
      MOVP    K32767 D9086
2574  LD      M7162  ; [PPID]  配方搜尋比對NG
      OR      M7163  ; [PPID]  配方搜尋比對NG(空白)
      MOVP    K0 D9086
2579  LDI     M7161  ; [PPID]  配方搜尋比對OK
      ANI     M7162  ; [PPID]  配方搜尋比對NG
      ANI     M7163  ; [PPID]  配方搜尋比對NG(空白)
      INV
      OUT     T2619 K5
2587  LD      T2619
      RST     M7161  ; [PPID]  配方搜尋比對OK
      RST     M7162  ; [PPID]  配方搜尋比對NG
      RST     M7163  ; [PPID]  配方搜尋比對NG(空白)
      RST     M7160  ; [PPID]  配方搜尋KP
2593  LD      SM402  ; Run Pls
      RST     M7062  ; 上位停止放板KP
2595  LD      M7205  ; 上位停止放板並清出料號
      OR      M7062  ; 上位停止放板KP
      ANI     M7204  ; 上位允許放板START
      AND     M6002  ; HMI-SECS- 通訊連線LAMP
      AND     M6006  ; HMI-PB  SECS  遠程/本地
      OUT     M7062  ; 上位停止放板KP
2601  LD      M7209  ; 上位下暫停進板
      OR      M8035
      ANI     M7210  ; 上位下恢復進板
      OUT     M8035
2605  LD      M7218  ; 和上位連線中
      LD      M7204  ; 上位允許放板START
      OR      M8034  ; 上位允許放板START KP
      ANB
      ANI     M7205  ; 上位停止放板並清出料號
      ANI     M6101  ; 回上位SECS控制模式切換
      OUT     M8034  ; 上位允許放板START KP
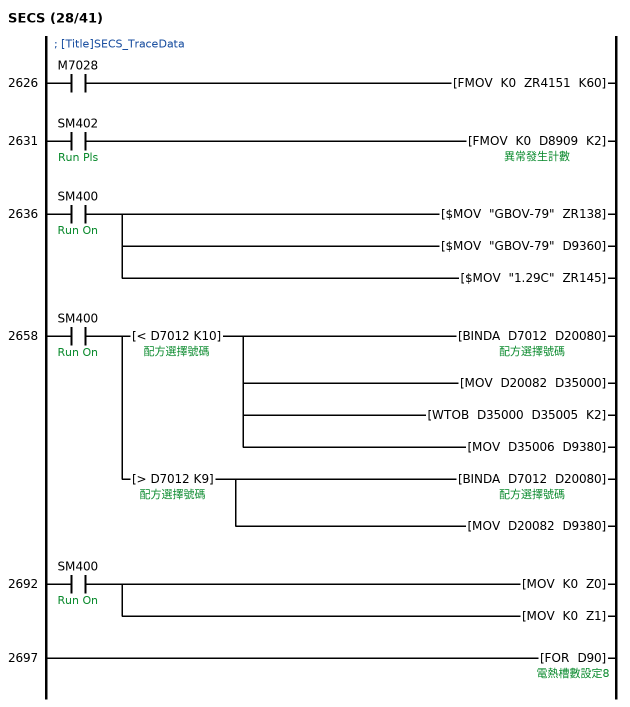
; [Title]SECS_TraceData
2626  LD      M7028
      FMOV    K0 ZR4151 K60
2631  LD      SM402  ; Run Pls
      FMOV    K0 D8909 K2  ; 異常發生計數
2636  LD      SM400  ; Run On
      $MOV    "GBOV-79" ZR138
      $MOV    "GBOV-79" D9360
      $MOV    "1.29C" ZR145
2658  LD      SM400  ; Run On
      MPS
      AND<    D7012 K10  ; 配方選擇號碼
      BINDA   D7012 D20080
      MOV     D20082 D35000
      WTOB    D35000 D35005 K2
      MOV     D35006 D9380
      MPP
      AND>    D7012 K9  ; 配方選擇號碼
      BINDA   D7012 D20080
      MOV     D20082 D9380
2692  LD      SM400  ; Run On
      MOV     K0 Z0
      MOV     K0 Z1
2697  FOR     D90  ; 電熱槽數設定8
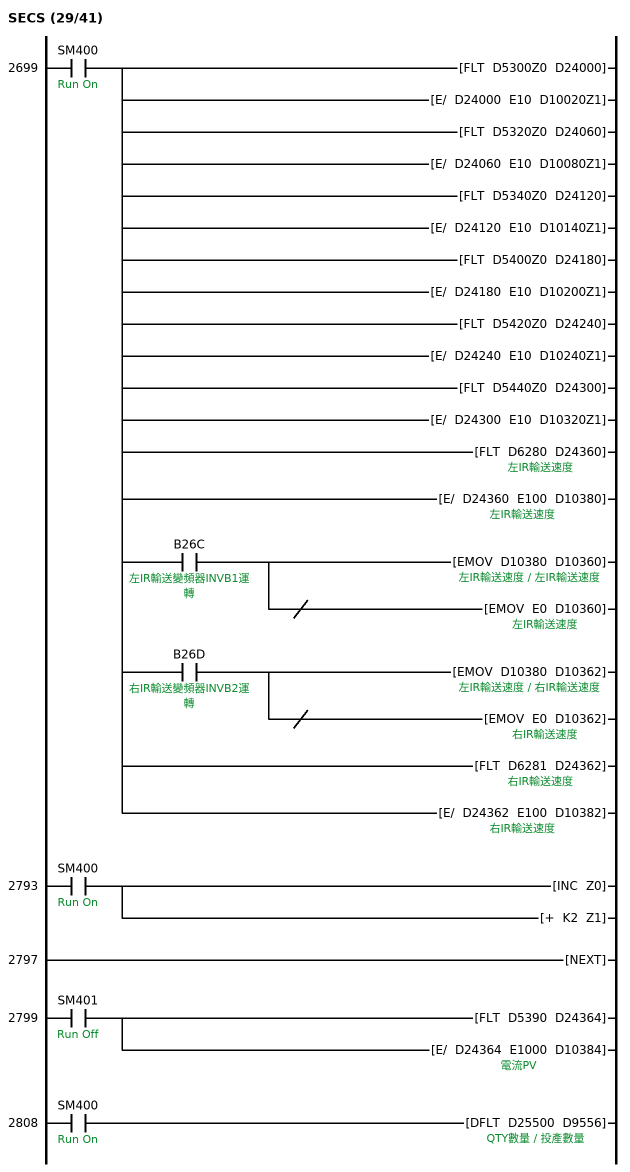
2699  LD      SM400  ; Run On
      FLT     D5300Z0 D24000
      E/      D24000 E10 D10020Z1
      FLT     D5320Z0 D24060
      E/      D24060 E10 D10080Z1
      FLT     D5340Z0 D24120
      E/      D24120 E10 D10140Z1
      FLT     D5400Z0 D24180
      E/      D24180 E10 D10200Z1
      FLT     D5420Z0 D24240
      E/      D24240 E10 D10240Z1
      FLT     D5440Z0 D24300
      E/      D24300 E10 D10320Z1
      FLT     D6280 D24360  ; 左IR輸送速度
      E/      D24360 E100 D10380  ; 左IR輸送速度
      MPS
      AND     B26C  ; 左IR輸送變頻器INVB1運轉
      EMOV    D10380 D10360  ; 左IR輸送速度
      INV
      EMOV    E0 D10360
      MRD
      AND     B26D  ; 右IR輸送變頻器INVB2運轉
      EMOV    D10380 D10362  ; 右IR輸送速度
      INV
      EMOV    E0 D10362
      MPP
      FLT     D6281 D24362  ; 右IR輸送速度
      E/      D24362 E100 D10382  ; 右IR輸送速度
2793  LD      SM400  ; Run On
      INC     Z0
      +       K2 Z1
2797  NEXT
2799  LD      SM401  ; Run Off
      FLT     D5390 D24364
      E/      D24364 E1000 D10384  ; 電流PV
2808  LD      SM400  ; Run On
      DFLT    D25500 D9556  ; 投產數量
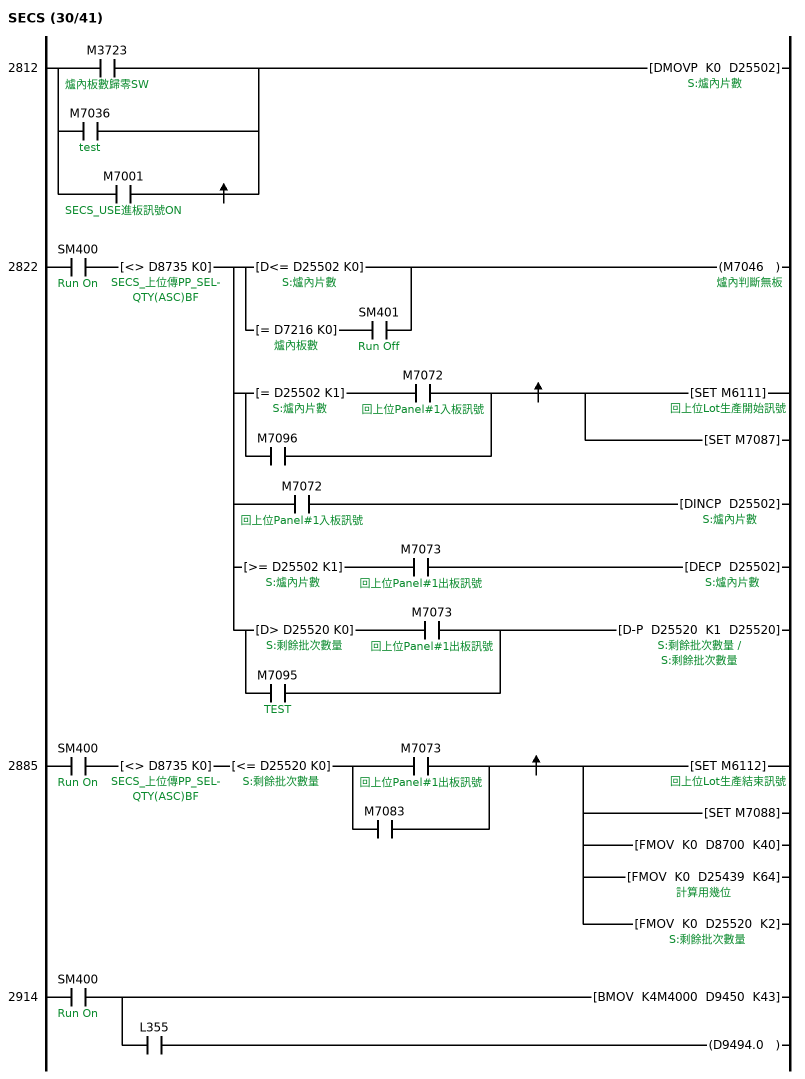
2812  LD      M3723  ; 爐內板數歸零SW
      OR      M7036  ; test
      LD      M7001  ; SECS_USE進板訊號ON
      MEP
      ORB
      DMOVP   K0 D25502  ; S:爐內片數
2822  LD      SM400  ; Run On
      AND<>   D8735 K0  ; SECS_上位傳PP_SEL-QTY(ASC)BF
      MPS
      LDD<=   D25502 K0  ; S:爐內片數
      LD=     D7216 K0  ; 爐內板數
      AND     SM401  ; Run Off
      ORB
      ANB
      OUT     M7046  ; 爐內判斷無板
      MRD
      LD=     D25502 K1  ; S:爐內片數
      AND     M7072  ; 回上位Panel#1入板訊號
      OR      M7096
      ANB
      MEP
      SET     M6111  ; 回上位Lot生產開始訊號
      SET     M7087
      MRD
      AND     M7072  ; 回上位Panel#1入板訊號
      DINCP   D25502
      MRD
      AND>=   D25502 K1  ; S:爐內片數
      AND     M7073  ; 回上位Panel#1出板訊號
      DECP    D25502
      MPP
      LDD>    D25520 K0  ; S:剩餘批次數量
      AND     M7073  ; 回上位Panel#1出板訊號
      OR      M7095  ; TEST
      ANB
      D-P     D25520 K1 D25520
2885  LD      SM400  ; Run On
      AND<>   D8735 K0  ; SECS_上位傳PP_SEL-QTY(ASC)BF
      AND<=   D25520 K0  ; S:剩餘批次數量
      LD      M7073  ; 回上位Panel#1出板訊號
      OR      M7083
      ANB
      MEP
      SET     M6112  ; 回上位Lot生產結束訊號
      SET     M7088
      FMOV    K0 D8700 K40
      FMOV    K0 D25439 K64
      FMOV    K0 D25520 K2
2914  LD      SM400  ; Run On
      BMOV    K4M4000 D9450 K43  ; 緊急停止
      AND     L355
      OUT     D9494.0
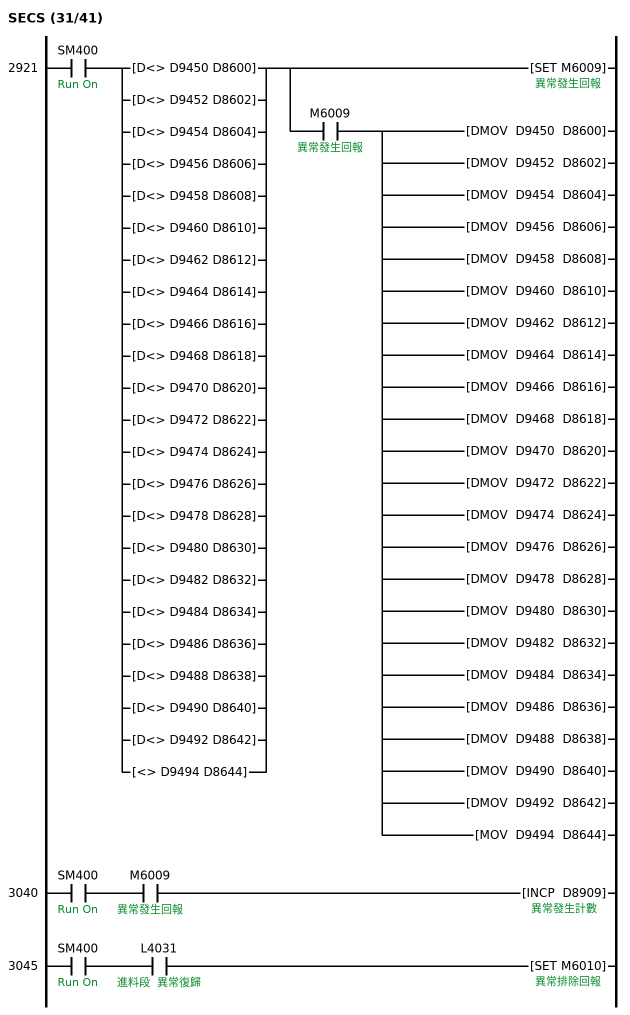
2921  LD      SM400  ; Run On
      LDD<>   D9450 D8600
      ORD<>   D9452 D8602
      ORD<>   D9454 D8604
      ORD<>   D9456 D8606
      ORD<>   D9458 D8608
      ORD<>   D9460 D8610
      ORD<>   D9462 D8612
      ORD<>   D9464 D8614
      ORD<>   D9466 D8616
      ORD<>   D9468 D8618
      ORD<>   D9470 D8620
      ORD<>   D9472 D8622
      ORD<>   D9474 D8624
      ORD<>   D9476 D8626
      ORD<>   D9478 D8628
      ORD<>   D9480 D8630
      ORD<>   D9482 D8632
      ORD<>   D9484 D8634
      ORD<>   D9486 D8636
      ORD<>   D9488 D8638
      ORD<>   D9490 D8640
      ORD<>   D9492 D8642
      OR<>    D9494 D8644
      ANB
      SET     M6009  ; 異常發生回報
      AND     M6009  ; 異常發生回報
      DMOV    D9450 D8600
      DMOV    D9452 D8602
      DMOV    D9454 D8604
      DMOV    D9456 D8606
      DMOV    D9458 D8608
      DMOV    D9460 D8610
      DMOV    D9462 D8612
      DMOV    D9464 D8614
      DMOV    D9466 D8616
      DMOV    D9468 D8618
      DMOV    D9470 D8620
      DMOV    D9472 D8622
      DMOV    D9474 D8624
      DMOV    D9476 D8626
      DMOV    D9478 D8628
      DMOV    D9480 D8630
      DMOV    D9482 D8632
      DMOV    D9484 D8634
      DMOV    D9486 D8636
      DMOV    D9488 D8638
      DMOV    D9490 D8640
      DMOV    D9492 D8642
      MOV     D9494 D8644
3040  LD      SM400  ; Run On
      AND     M6009  ; 異常發生回報
      INCP    D8909
3045  LD      SM400  ; Run On
      AND     L4031  ; 進料段  異常復歸
      SET     M6010  ; 異常排除回報
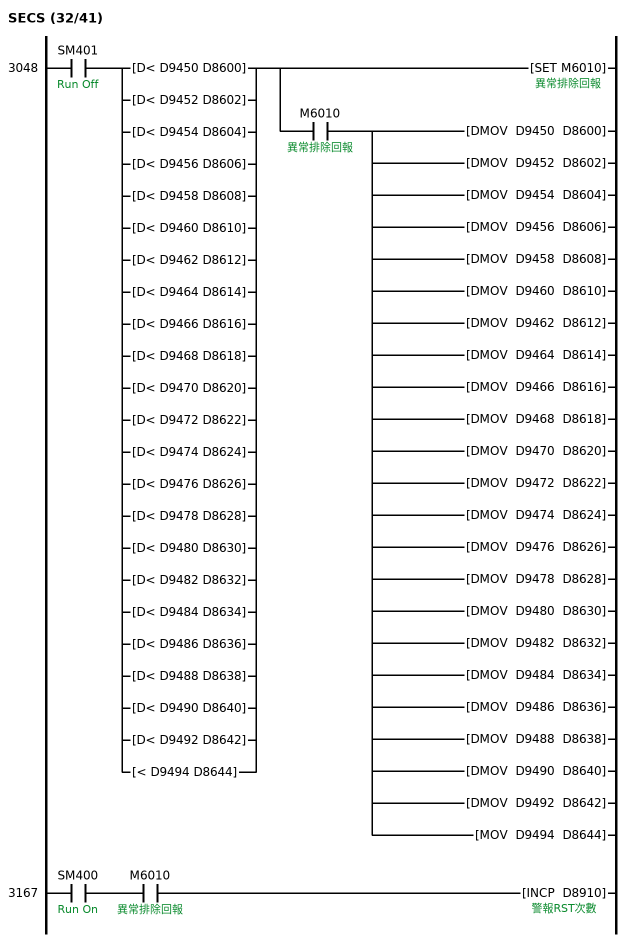
3048  LD      SM401  ; Run Off
      LDD<    D9450 D8600
      ORD<    D9452 D8602
      ORD<    D9454 D8604
      ORD<    D9456 D8606
      ORD<    D9458 D8608
      ORD<    D9460 D8610
      ORD<    D9462 D8612
      ORD<    D9464 D8614
      ORD<    D9466 D8616
      ORD<    D9468 D8618
      ORD<    D9470 D8620
      ORD<    D9472 D8622
      ORD<    D9474 D8624
      ORD<    D9476 D8626
      ORD<    D9478 D8628
      ORD<    D9480 D8630
      ORD<    D9482 D8632
      ORD<    D9484 D8634
      ORD<    D9486 D8636
      ORD<    D9488 D8638
      ORD<    D9490 D8640
      ORD<    D9492 D8642
      OR<     D9494 D8644
      ANB
      SET     M6010  ; 異常排除回報
      AND     M6010  ; 異常排除回報
      DMOV    D9450 D8600
      DMOV    D9452 D8602
      DMOV    D9454 D8604
      DMOV    D9456 D8606
      DMOV    D9458 D8608
      DMOV    D9460 D8610
      DMOV    D9462 D8612
      DMOV    D9464 D8614
      DMOV    D9466 D8616
      DMOV    D9468 D8618
      DMOV    D9470 D8620
      DMOV    D9472 D8622
      DMOV    D9474 D8624
      DMOV    D9476 D8626
      DMOV    D9478 D8628
      DMOV    D9480 D8630
      DMOV    D9482 D8632
      DMOV    D9484 D8634
      DMOV    D9486 D8636
      DMOV    D9488 D8638
      DMOV    D9490 D8640
      DMOV    D9492 D8642
      MOV     D9494 D8644
3167  LD      SM400  ; Run On
      AND     M6010  ; 異常排除回報
      INCP    D8910  ; 警報RST次數
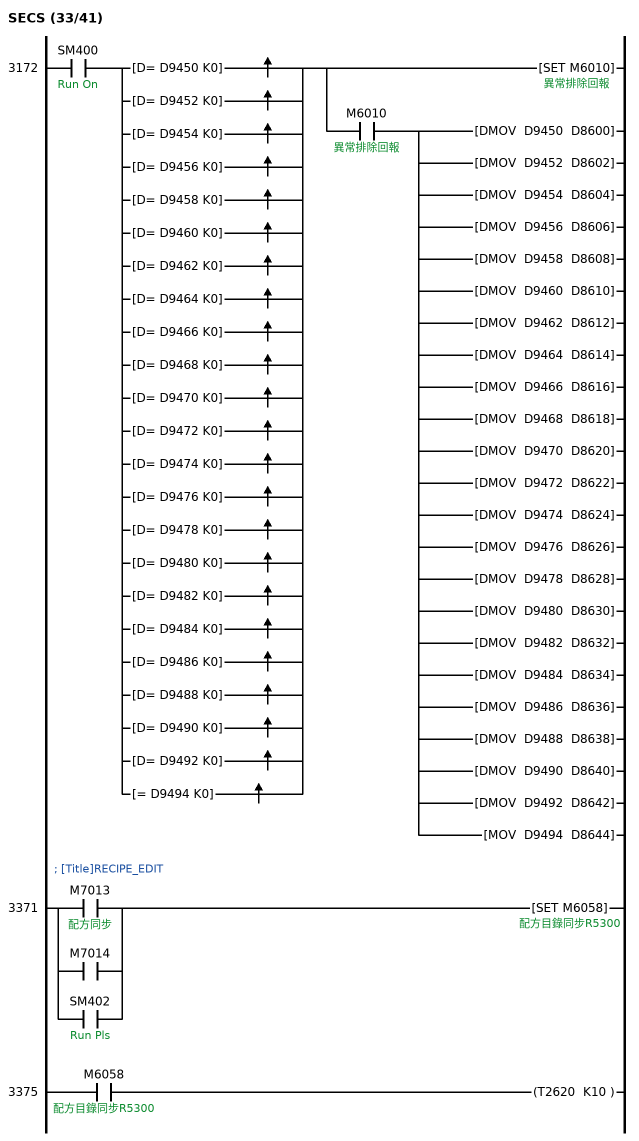
3172  LD      SM400  ; Run On
      LDD=    D9450 K0
      MEP
      LDD=    D9452 K0
      MEP
      ORB
      LDD=    D9454 K0
      MEP
      ORB
      LDD=    D9456 K0
      MEP
      ORB
      LDD=    D9458 K0
      MEP
      ORB
      LDD=    D9460 K0
      MEP
      ORB
      LDD=    D9462 K0
      MEP
      ORB
      LDD=    D9464 K0
      MEP
      ORB
      LDD=    D9466 K0
      MEP
      ORB
      LDD=    D9468 K0
      MEP
      ORB
      LDD=    D9470 K0
      MEP
      ORB
      LDD=    D9472 K0
      MEP
      ORB
      LDD=    D9474 K0
      MEP
      ORB
      LDD=    D9476 K0
      MEP
      ORB
      LDD=    D9478 K0
      MEP
      ORB
      LDD=    D9480 K0
      MEP
      ORB
      LDD=    D9482 K0
      MEP
      ORB
      LDD=    D9484 K0
      MEP
      ORB
      LDD=    D9486 K0
      MEP
      ORB
      LDD=    D9488 K0
      MEP
      ORB
      LDD=    D9490 K0
      MEP
      ORB
      LDD=    D9492 K0
      MEP
      ORB
      LD=     D9494 K0
      MEP
      ORB
      ANB
      SET     M6010  ; 異常排除回報
      AND     M6010  ; 異常排除回報
      DMOV    D9450 D8600
      DMOV    D9452 D8602
      DMOV    D9454 D8604
      DMOV    D9456 D8606
      DMOV    D9458 D8608
      DMOV    D9460 D8610
      DMOV    D9462 D8612
      DMOV    D9464 D8614
      DMOV    D9466 D8616
      DMOV    D9468 D8618
      DMOV    D9470 D8620
      DMOV    D9472 D8622
      DMOV    D9474 D8624
      DMOV    D9476 D8626
      DMOV    D9478 D8628
      DMOV    D9480 D8630
      DMOV    D9482 D8632
      DMOV    D9484 D8634
      DMOV    D9486 D8636
      DMOV    D9488 D8638
      DMOV    D9490 D8640
      DMOV    D9492 D8642
      MOV     D9494 D8644
; [Title]RECIPE_EDIT
3371  LD      M7013  ; 配方同步
      OR      M7014
      OR      SM402  ; Run Pls
      SET     M6058  ; 配方目錄同步R5300
3375  LD      M6058  ; 配方目錄同步R5300
      OUT     T2620 K10
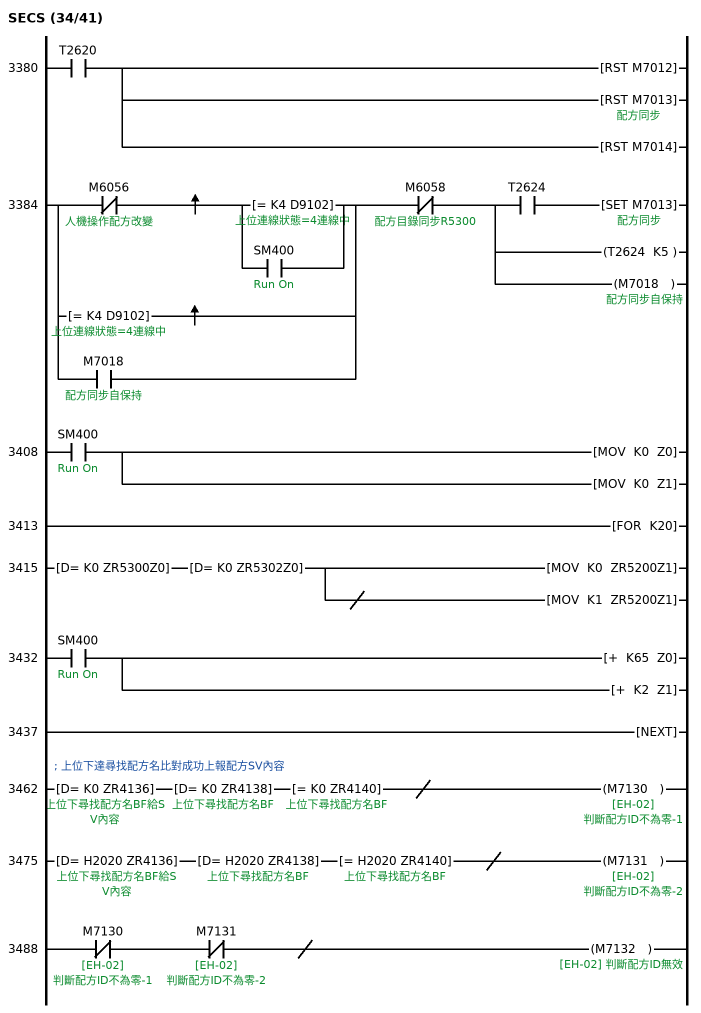
3380  LD      T2620
      RST     M7012
      RST     M7013  ; 配方同步
      RST     M7014
3384  LDI     M6056  ; 人機操作配方改變
      MEP
      LD=     K4 D9102  ; 上位連線狀態=4連線中
      OR      SM400  ; Run On
      ANB
      LD=     K4 D9102  ; 上位連線狀態=4連線中
      MEP
      ORB
      OR      M7018  ; 配方同步自保持
      ANI     M6058  ; 配方目錄同步R5300
      MPS
      AND     T2624
      SET     M7013  ; 配方同步
      MPP
      OUT     T2624 K5
      OUT     M7018  ; 配方同步自保持
3408  LD      SM400  ; Run On
      MOV     K0 Z0
      MOV     K0 Z1
3413  FOR     K20
3415  LDD=    K0 ZR5300Z0
      ANDD=   K0 ZR5302Z0
      MOV     K0 ZR5200Z1
      INV
      MOV     K1 ZR5200Z1
3432  LD      SM400  ; Run On
      +       K65 Z0
      +       K2 Z1
3437  NEXT
; 上位下達尋找配方名比對成功上報配方SV內容
3462  LDD=    K0 ZR4136  ; 上位下尋找配方名BF給SV內容
      ANDD=   K0 ZR4138  ; 上位下尋找配方名BF
      AND=    K0 ZR4140  ; 上位下尋找配方名BF
      INV
      OUT     M7130  ; [EH-02] 判斷配方ID不為零-1
3475  LDD=    H2020 ZR4136  ; 上位下尋找配方名BF給SV內容
      ANDD=   H2020 ZR4138  ; 上位下尋找配方名BF
      AND=    H2020 ZR4140  ; 上位下尋找配方名BF
      INV
      OUT     M7131  ; [EH-02] 判斷配方ID不為零-2
3488  LDI     M7130  ; [EH-02] 判斷配方ID不為零-1
      ANI     M7131  ; [EH-02] 判斷配方ID不為零-2
      INV
      OUT     M7132  ; [EH-02] 判斷配方ID無效
